// TIA Portal V17 export
// export: Created 2025-03-10T12:15:34.5959597Z, ExportSetting WithDefaults, DisplayName Totally Integrated Automation Portal, DisplayVersion V17 Update 8, DisplayName TIA Portal Openness, DisplayVersion V17 Update 8, DisplayName TIA Portal Version Control Interface, DisplayVersion V17, DisplayName SINAMICS Startdrive Advanced, DisplayVersion V17 SP2, DisplayName SINAMICS Startdrive G110M, G120, G120C, G120D, G120P, G115D, DisplayVersion V17 SP2, DisplayName SINAMICS Startdrive G130, G150, S120, S150, SINAMICS MV, S210, DisplayVersion V17 SP2, DisplayName STEP 7 Professional, DisplayVersion V17 Update 8, DisplayName SINUMERIK ONE STEP 7 Toolbox, DisplayVersion V17 Update 12, DisplayName SINUMERIK 840D sl STEP 7 Toolbox, DisplayVersion V17 Update 12, DisplayName STEP 7 Safety, DisplayVersion V17 Update 6, DisplayName WinCC Advanced, DisplayVersion V17 Update 8
FUNCTION "FC369_NCK_M_CH8_UNIT_03" : Void   // FC369, LAD
TITLE = Channel 1 data
{ S7_Optimized_Access := 'FALSE' }
AUTHOR : ETXETAR
VERSION : 1.0
// stored: AutoNumber false, IsIECCheckEnabled false, SetENOAutomatically false, UDAEnableTagReadback false
BEGIN

REGION Network 1: ACKNOWLEDGE M400-FIXTURE 1 CLAMP SEQUENCE (READ-IN DISABLE) / ACKNOWLEDGE M100-CLAMP SEQUENCE FIXTURE 1
   // NOTE: WHEN THERE IS NOT INDEXING TABLE AVAILABLE IN THE MACHINE DELETE 
   // DB2171.DBX5.0 AND DB2171.DBX2.0
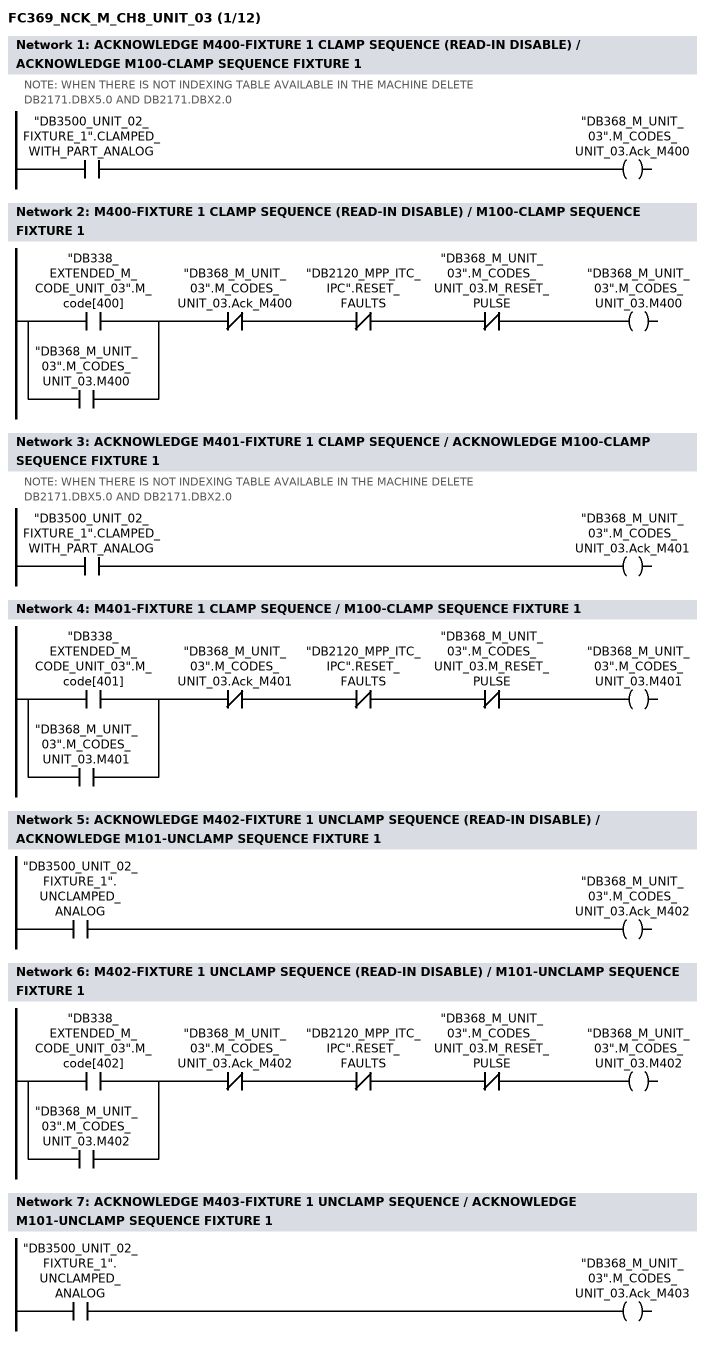
   RUNG wire#powerrail
      Contact( "DB3500_UNIT_02_FIXTURE_1".CLAMPED_WITH_PART_ANALOG )
      Coil( "DB368_M_UNIT_03".M_CODES_UNIT_03.Ack_M400 )
   END_RUNG
   // the same network as SCL:
   "DB368_M_UNIT_03".M_CODES_UNIT_03.Ack_M400 := "DB3500_UNIT_02_FIXTURE_1".CLAMPED_WITH_PART_ANALOG;
END_REGION

REGION Network 2: M400-FIXTURE 1 CLAMP SEQUENCE (READ-IN DISABLE) / M100-CLAMP SEQUENCE FIXTURE 1
   RUNG wire#powerrail
      Contact( "DB338_EXTENDED_M_CODE_UNIT_03".M_code[400] )
      wire#w1
      I_Contact( "DB368_M_UNIT_03".M_CODES_UNIT_03.Ack_M400 )
      I_Contact( "DB2120_MPP_ITC_IPC".RESET_FAULTS )
      I_Contact( "DB368_M_UNIT_03".M_CODES_UNIT_03.M_RESET_PULSE )
      Coil( "DB368_M_UNIT_03".M_CODES_UNIT_03.M400 )
   END_RUNG
   RUNG wire#powerrail
      Contact( "DB368_M_UNIT_03".M_CODES_UNIT_03.M400 )
   END_RUNG wire#w1
   // the same network as SCL:
   "DB368_M_UNIT_03".M_CODES_UNIT_03.M400 := ("DB338_EXTENDED_M_CODE_UNIT_03".M_code[400] OR "DB368_M_UNIT_03".M_CODES_UNIT_03.M400) AND NOT "DB368_M_UNIT_03".M_CODES_UNIT_03.Ack_M400 AND NOT "DB2120_MPP_ITC_IPC".RESET_FAULTS AND NOT "DB368_M_UNIT_03".M_CODES_UNIT_03.M_RESET_PULSE;
END_REGION

REGION Network 3: ACKNOWLEDGE M401-FIXTURE 1 CLAMP SEQUENCE / ACKNOWLEDGE M100-CLAMP SEQUENCE FIXTURE 1
   // NOTE: WHEN THERE IS NOT INDEXING TABLE AVAILABLE IN THE MACHINE DELETE 
   // DB2171.DBX5.0 AND DB2171.DBX2.0
   RUNG wire#powerrail
      Contact( "DB3500_UNIT_02_FIXTURE_1".CLAMPED_WITH_PART_ANALOG )
      Coil( "DB368_M_UNIT_03".M_CODES_UNIT_03.Ack_M401 )
   END_RUNG
   // the same network as SCL:
   "DB368_M_UNIT_03".M_CODES_UNIT_03.Ack_M401 := "DB3500_UNIT_02_FIXTURE_1".CLAMPED_WITH_PART_ANALOG;
END_REGION

REGION Network 4: M401-FIXTURE 1 CLAMP SEQUENCE / M100-CLAMP SEQUENCE FIXTURE 1
   RUNG wire#powerrail
      Contact( "DB338_EXTENDED_M_CODE_UNIT_03".M_code[401] )
      wire#w1
      I_Contact( "DB368_M_UNIT_03".M_CODES_UNIT_03.Ack_M401 )
      I_Contact( "DB2120_MPP_ITC_IPC".RESET_FAULTS )
      I_Contact( "DB368_M_UNIT_03".M_CODES_UNIT_03.M_RESET_PULSE )
      Coil( "DB368_M_UNIT_03".M_CODES_UNIT_03.M401 )
   END_RUNG
   RUNG wire#powerrail
      Contact( "DB368_M_UNIT_03".M_CODES_UNIT_03.M401 )
   END_RUNG wire#w1
   // the same network as SCL:
   "DB368_M_UNIT_03".M_CODES_UNIT_03.M401 := ("DB338_EXTENDED_M_CODE_UNIT_03".M_code[401] OR "DB368_M_UNIT_03".M_CODES_UNIT_03.M401) AND NOT "DB368_M_UNIT_03".M_CODES_UNIT_03.Ack_M401 AND NOT "DB2120_MPP_ITC_IPC".RESET_FAULTS AND NOT "DB368_M_UNIT_03".M_CODES_UNIT_03.M_RESET_PULSE;
END_REGION

REGION Network 5: ACKNOWLEDGE M402-FIXTURE 1 UNCLAMP SEQUENCE (READ-IN DISABLE) / ACKNOWLEDGE M101-UNCLAMP SEQUENCE FIXTURE 1
   RUNG wire#powerrail
      Contact( "DB3500_UNIT_02_FIXTURE_1".UNCLAMPED_ANALOG )
      Coil( "DB368_M_UNIT_03".M_CODES_UNIT_03.Ack_M402 )
   END_RUNG
   // the same network as SCL:
   "DB368_M_UNIT_03".M_CODES_UNIT_03.Ack_M402 := "DB3500_UNIT_02_FIXTURE_1".UNCLAMPED_ANALOG;
END_REGION

REGION Network 6: M402-FIXTURE 1 UNCLAMP SEQUENCE (READ-IN DISABLE) / M101-UNCLAMP SEQUENCE FIXTURE 1
   RUNG wire#powerrail
      Contact( "DB338_EXTENDED_M_CODE_UNIT_03".M_code[402] )
      wire#w1
      I_Contact( "DB368_M_UNIT_03".M_CODES_UNIT_03.Ack_M402 )
      I_Contact( "DB2120_MPP_ITC_IPC".RESET_FAULTS )
      I_Contact( "DB368_M_UNIT_03".M_CODES_UNIT_03.M_RESET_PULSE )
      Coil( "DB368_M_UNIT_03".M_CODES_UNIT_03.M402 )
   END_RUNG
   RUNG wire#powerrail
      Contact( "DB368_M_UNIT_03".M_CODES_UNIT_03.M402 )
   END_RUNG wire#w1
   // the same network as SCL:
   "DB368_M_UNIT_03".M_CODES_UNIT_03.M402 := ("DB338_EXTENDED_M_CODE_UNIT_03".M_code[402] OR "DB368_M_UNIT_03".M_CODES_UNIT_03.M402) AND NOT "DB368_M_UNIT_03".M_CODES_UNIT_03.Ack_M402 AND NOT "DB2120_MPP_ITC_IPC".RESET_FAULTS AND NOT "DB368_M_UNIT_03".M_CODES_UNIT_03.M_RESET_PULSE;
END_REGION

REGION Network 7: ACKNOWLEDGE M403-FIXTURE 1 UNCLAMP SEQUENCE / ACKNOWLEDGE M101-UNCLAMP SEQUENCE FIXTURE 1
   RUNG wire#powerrail
      Contact( "DB3500_UNIT_02_FIXTURE_1".UNCLAMPED_ANALOG )
      Coil( "DB368_M_UNIT_03".M_CODES_UNIT_03.Ack_M403 )
   END_RUNG
   // the same network as SCL:
   "DB368_M_UNIT_03".M_CODES_UNIT_03.Ack_M403 := "DB3500_UNIT_02_FIXTURE_1".UNCLAMPED_ANALOG;
END_REGION

REGION Network 8: M403-FIXTURE 1 UNCLAMP SEQUENCE / M101-UNCLAMP SEQUENCE FIXTURE 1
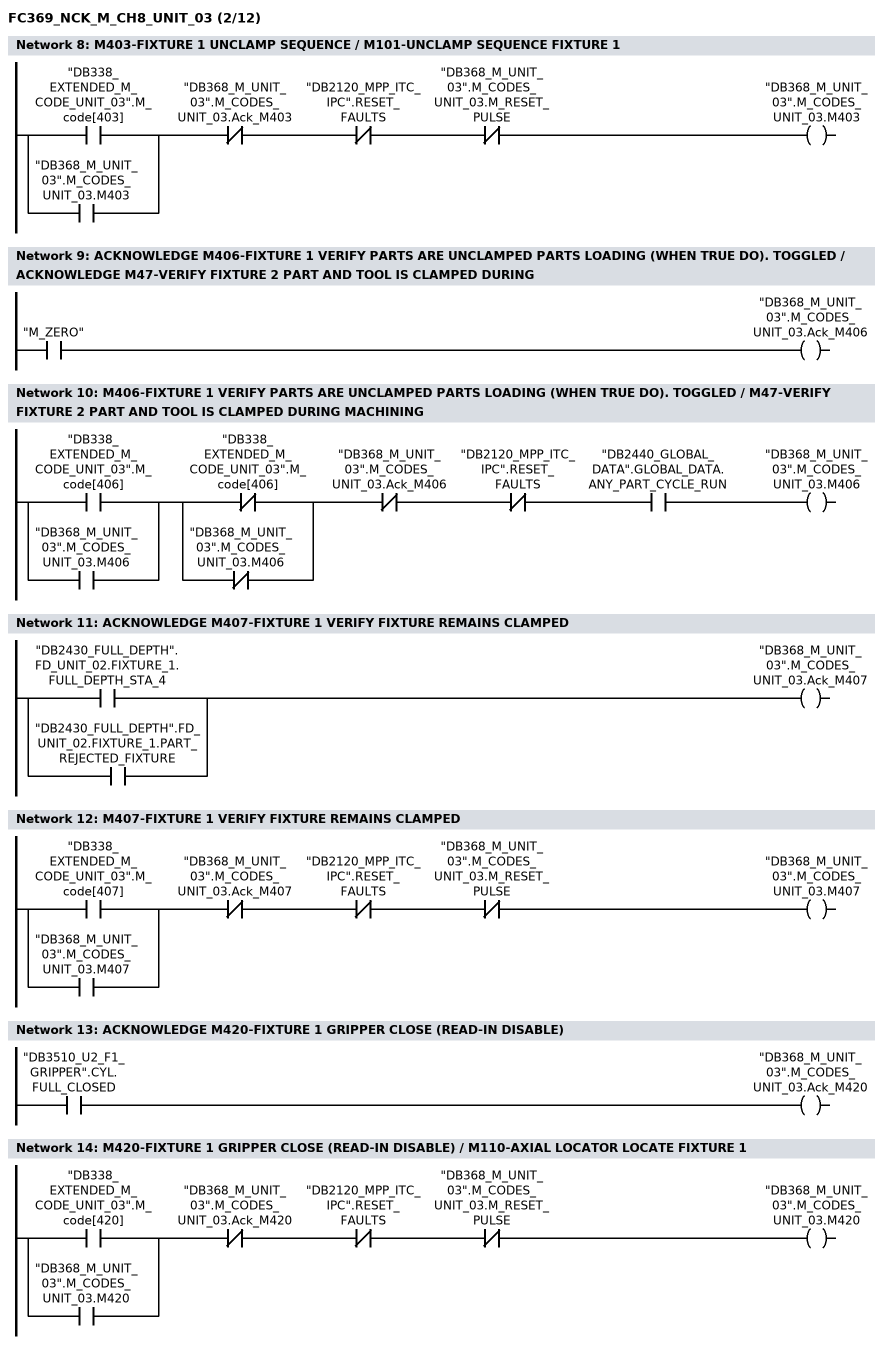
   RUNG wire#powerrail
      Contact( "DB338_EXTENDED_M_CODE_UNIT_03".M_code[403] )
      wire#w1
      I_Contact( "DB368_M_UNIT_03".M_CODES_UNIT_03.Ack_M403 )
      I_Contact( "DB2120_MPP_ITC_IPC".RESET_FAULTS )
      I_Contact( "DB368_M_UNIT_03".M_CODES_UNIT_03.M_RESET_PULSE )
      Coil( "DB368_M_UNIT_03".M_CODES_UNIT_03.M403 )
   END_RUNG
   RUNG wire#powerrail
      Contact( "DB368_M_UNIT_03".M_CODES_UNIT_03.M403 )
   END_RUNG wire#w1
   // the same network as SCL:
   "DB368_M_UNIT_03".M_CODES_UNIT_03.M403 := ("DB338_EXTENDED_M_CODE_UNIT_03".M_code[403] OR "DB368_M_UNIT_03".M_CODES_UNIT_03.M403) AND NOT "DB368_M_UNIT_03".M_CODES_UNIT_03.Ack_M403 AND NOT "DB2120_MPP_ITC_IPC".RESET_FAULTS AND NOT "DB368_M_UNIT_03".M_CODES_UNIT_03.M_RESET_PULSE;
END_REGION

REGION Network 9: ACKNOWLEDGE M406-FIXTURE 1 VERIFY PARTS ARE UNCLAMPED PARTS LOADING (WHEN TRUE DO). TOGGLED / ACKNOWLEDGE M47-VERIFY FIXTURE 2 PART AND TOOL IS CLAMPED DURING
   RUNG wire#powerrail
      Contact( "M_ZERO" )
      Coil( "DB368_M_UNIT_03".M_CODES_UNIT_03.Ack_M406 )
   END_RUNG
   // the same network as SCL:
   "DB368_M_UNIT_03".M_CODES_UNIT_03.Ack_M406 := "M_ZERO";
END_REGION

REGION Network 10: M406-FIXTURE 1 VERIFY PARTS ARE UNCLAMPED PARTS LOADING (WHEN TRUE DO). TOGGLED / M47-VERIFY FIXTURE 2 PART AND TOOL IS CLAMPED DURING MACHINING
   RUNG wire#powerrail
      Contact( "DB338_EXTENDED_M_CODE_UNIT_03".M_code[406] )
      wire#w1
      I_Contact( "DB338_EXTENDED_M_CODE_UNIT_03".M_code[406] )
      wire#w2
      I_Contact( "DB368_M_UNIT_03".M_CODES_UNIT_03.Ack_M406 )
      I_Contact( "DB2120_MPP_ITC_IPC".RESET_FAULTS )
      Contact( "DB2440_GLOBAL_DATA".GLOBAL_DATA.ANY_PART_CYCLE_RUN )
      Coil( "DB368_M_UNIT_03".M_CODES_UNIT_03.M406 )
   END_RUNG
   RUNG wire#powerrail
      Contact( "DB368_M_UNIT_03".M_CODES_UNIT_03.M406 )
   END_RUNG wire#w1
   RUNG wire#w1
      I_Contact( "DB368_M_UNIT_03".M_CODES_UNIT_03.M406 )
   END_RUNG wire#w2
   // the same network as SCL:
   "DB368_M_UNIT_03".M_CODES_UNIT_03.M406 := ("DB338_EXTENDED_M_CODE_UNIT_03".M_code[406] OR "DB368_M_UNIT_03".M_CODES_UNIT_03.M406) AND (NOT "DB338_EXTENDED_M_CODE_UNIT_03".M_code[406] OR NOT "DB368_M_UNIT_03".M_CODES_UNIT_03.M406) AND NOT "DB368_M_UNIT_03".M_CODES_UNIT_03.Ack_M406 AND NOT "DB2120_MPP_ITC_IPC".RESET_FAULTS AND "DB2440_GLOBAL_DATA".GLOBAL_DATA.ANY_PART_CYCLE_RUN;
END_REGION

REGION Network 11: ACKNOWLEDGE M407-FIXTURE 1 VERIFY FIXTURE REMAINS CLAMPED
   RUNG wire#powerrail
      Contact( "DB2430_FULL_DEPTH".FD_UNIT_02.FIXTURE_1.FULL_DEPTH_STA_4 )
      wire#w1
      Coil( "DB368_M_UNIT_03".M_CODES_UNIT_03.Ack_M407 )
   END_RUNG
   RUNG wire#powerrail
      Contact( "DB2430_FULL_DEPTH".FD_UNIT_02.FIXTURE_1.PART_REJECTED_FIXTURE )
   END_RUNG wire#w1
   // the same network as SCL:
   "DB368_M_UNIT_03".M_CODES_UNIT_03.Ack_M407 := "DB2430_FULL_DEPTH".FD_UNIT_02.FIXTURE_1.FULL_DEPTH_STA_4 OR "DB2430_FULL_DEPTH".FD_UNIT_02.FIXTURE_1.PART_REJECTED_FIXTURE;
END_REGION

REGION Network 12: M407-FIXTURE 1 VERIFY FIXTURE REMAINS CLAMPED
   RUNG wire#powerrail
      Contact( "DB338_EXTENDED_M_CODE_UNIT_03".M_code[407] )
      wire#w1
      I_Contact( "DB368_M_UNIT_03".M_CODES_UNIT_03.Ack_M407 )
      I_Contact( "DB2120_MPP_ITC_IPC".RESET_FAULTS )
      I_Contact( "DB368_M_UNIT_03".M_CODES_UNIT_03.M_RESET_PULSE )
      Coil( "DB368_M_UNIT_03".M_CODES_UNIT_03.M407 )
   END_RUNG
   RUNG wire#powerrail
      Contact( "DB368_M_UNIT_03".M_CODES_UNIT_03.M407 )
   END_RUNG wire#w1
   // the same network as SCL:
   "DB368_M_UNIT_03".M_CODES_UNIT_03.M407 := ("DB338_EXTENDED_M_CODE_UNIT_03".M_code[407] OR "DB368_M_UNIT_03".M_CODES_UNIT_03.M407) AND NOT "DB368_M_UNIT_03".M_CODES_UNIT_03.Ack_M407 AND NOT "DB2120_MPP_ITC_IPC".RESET_FAULTS AND NOT "DB368_M_UNIT_03".M_CODES_UNIT_03.M_RESET_PULSE;
END_REGION

REGION Network 13: ACKNOWLEDGE M420-FIXTURE 1 GRIPPER CLOSE (READ-IN DISABLE)
   RUNG wire#powerrail
      Contact( "DB3510_U2_F1_GRIPPER".CYL.FULL_CLOSED )
      Coil( "DB368_M_UNIT_03".M_CODES_UNIT_03.Ack_M420 )
   END_RUNG
   // the same network as SCL:
   "DB368_M_UNIT_03".M_CODES_UNIT_03.Ack_M420 := "DB3510_U2_F1_GRIPPER".CYL.FULL_CLOSED;
END_REGION

REGION Network 14: M420-FIXTURE 1 GRIPPER CLOSE (READ-IN DISABLE) / M110-AXIAL LOCATOR LOCATE FIXTURE 1
   RUNG wire#powerrail
      Contact( "DB338_EXTENDED_M_CODE_UNIT_03".M_code[420] )
      wire#w1
      I_Contact( "DB368_M_UNIT_03".M_CODES_UNIT_03.Ack_M420 )
      I_Contact( "DB2120_MPP_ITC_IPC".RESET_FAULTS )
      I_Contact( "DB368_M_UNIT_03".M_CODES_UNIT_03.M_RESET_PULSE )
      Coil( "DB368_M_UNIT_03".M_CODES_UNIT_03.M420 )
   END_RUNG
   RUNG wire#powerrail
      Contact( "DB368_M_UNIT_03".M_CODES_UNIT_03.M420 )
   END_RUNG wire#w1
   // the same network as SCL:
   "DB368_M_UNIT_03".M_CODES_UNIT_03.M420 := ("DB338_EXTENDED_M_CODE_UNIT_03".M_code[420] OR "DB368_M_UNIT_03".M_CODES_UNIT_03.M420) AND NOT "DB368_M_UNIT_03".M_CODES_UNIT_03.Ack_M420 AND NOT "DB2120_MPP_ITC_IPC".RESET_FAULTS AND NOT "DB368_M_UNIT_03".M_CODES_UNIT_03.M_RESET_PULSE;
END_REGION

REGION Network 15: ACKNOWLEDGE M421-FIXTURE 1 GRIPPER CLOSE
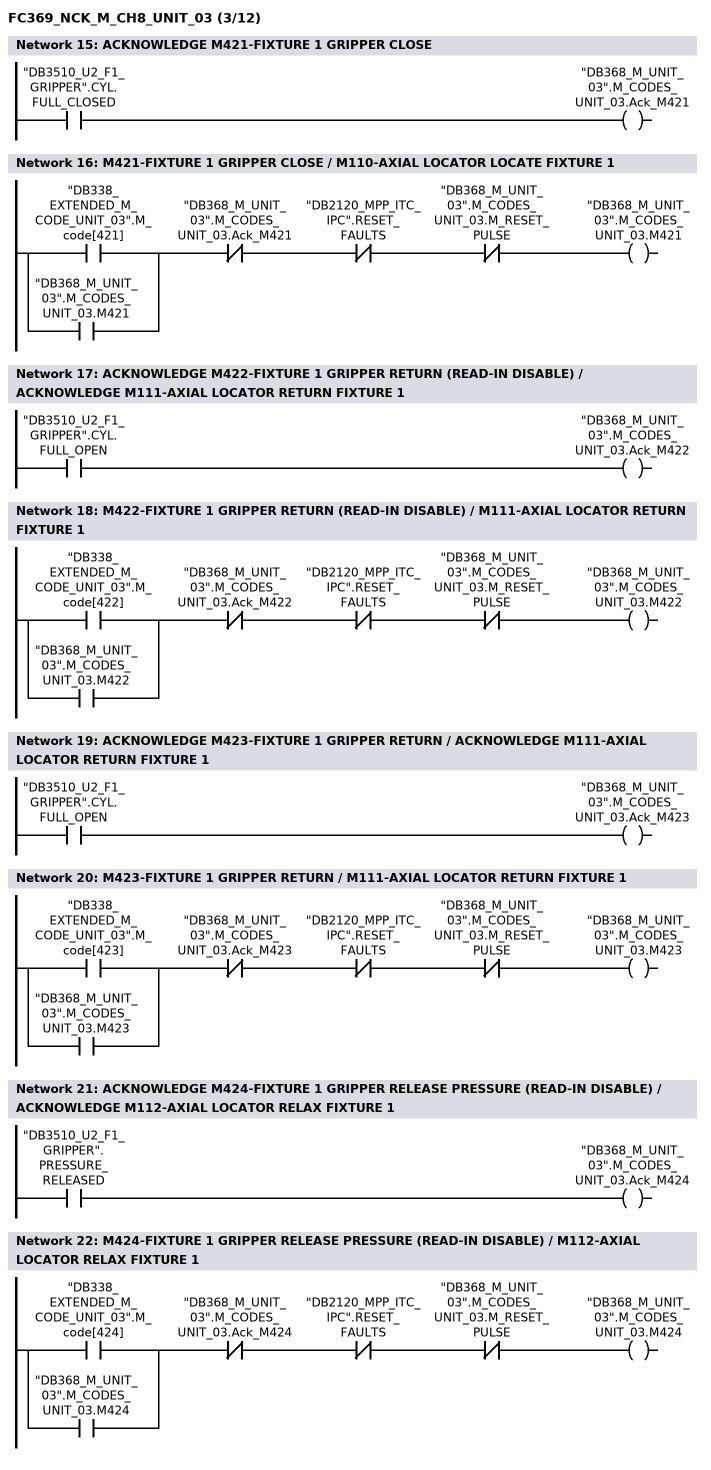
   RUNG wire#powerrail
      Contact( "DB3510_U2_F1_GRIPPER".CYL.FULL_CLOSED )
      Coil( "DB368_M_UNIT_03".M_CODES_UNIT_03.Ack_M421 )
   END_RUNG
   // the same network as SCL:
   "DB368_M_UNIT_03".M_CODES_UNIT_03.Ack_M421 := "DB3510_U2_F1_GRIPPER".CYL.FULL_CLOSED;
END_REGION

REGION Network 16: M421-FIXTURE 1 GRIPPER CLOSE / M110-AXIAL LOCATOR LOCATE FIXTURE 1
   RUNG wire#powerrail
      Contact( "DB338_EXTENDED_M_CODE_UNIT_03".M_code[421] )
      wire#w1
      I_Contact( "DB368_M_UNIT_03".M_CODES_UNIT_03.Ack_M421 )
      I_Contact( "DB2120_MPP_ITC_IPC".RESET_FAULTS )
      I_Contact( "DB368_M_UNIT_03".M_CODES_UNIT_03.M_RESET_PULSE )
      Coil( "DB368_M_UNIT_03".M_CODES_UNIT_03.M421 )
   END_RUNG
   RUNG wire#powerrail
      Contact( "DB368_M_UNIT_03".M_CODES_UNIT_03.M421 )
   END_RUNG wire#w1
   // the same network as SCL:
   "DB368_M_UNIT_03".M_CODES_UNIT_03.M421 := ("DB338_EXTENDED_M_CODE_UNIT_03".M_code[421] OR "DB368_M_UNIT_03".M_CODES_UNIT_03.M421) AND NOT "DB368_M_UNIT_03".M_CODES_UNIT_03.Ack_M421 AND NOT "DB2120_MPP_ITC_IPC".RESET_FAULTS AND NOT "DB368_M_UNIT_03".M_CODES_UNIT_03.M_RESET_PULSE;
END_REGION

REGION Network 17: ACKNOWLEDGE M422-FIXTURE 1 GRIPPER RETURN (READ-IN DISABLE) / ACKNOWLEDGE M111-AXIAL LOCATOR RETURN FIXTURE 1
   RUNG wire#powerrail
      Contact( "DB3510_U2_F1_GRIPPER".CYL.FULL_OPEN )
      Coil( "DB368_M_UNIT_03".M_CODES_UNIT_03.Ack_M422 )
   END_RUNG
   // the same network as SCL:
   "DB368_M_UNIT_03".M_CODES_UNIT_03.Ack_M422 := "DB3510_U2_F1_GRIPPER".CYL.FULL_OPEN;
END_REGION

REGION Network 18: M422-FIXTURE 1 GRIPPER RETURN (READ-IN DISABLE) / M111-AXIAL LOCATOR RETURN FIXTURE 1
   RUNG wire#powerrail
      Contact( "DB338_EXTENDED_M_CODE_UNIT_03".M_code[422] )
      wire#w1
      I_Contact( "DB368_M_UNIT_03".M_CODES_UNIT_03.Ack_M422 )
      I_Contact( "DB2120_MPP_ITC_IPC".RESET_FAULTS )
      I_Contact( "DB368_M_UNIT_03".M_CODES_UNIT_03.M_RESET_PULSE )
      Coil( "DB368_M_UNIT_03".M_CODES_UNIT_03.M422 )
   END_RUNG
   RUNG wire#powerrail
      Contact( "DB368_M_UNIT_03".M_CODES_UNIT_03.M422 )
   END_RUNG wire#w1
   // the same network as SCL:
   "DB368_M_UNIT_03".M_CODES_UNIT_03.M422 := ("DB338_EXTENDED_M_CODE_UNIT_03".M_code[422] OR "DB368_M_UNIT_03".M_CODES_UNIT_03.M422) AND NOT "DB368_M_UNIT_03".M_CODES_UNIT_03.Ack_M422 AND NOT "DB2120_MPP_ITC_IPC".RESET_FAULTS AND NOT "DB368_M_UNIT_03".M_CODES_UNIT_03.M_RESET_PULSE;
END_REGION

REGION Network 19: ACKNOWLEDGE M423-FIXTURE 1 GRIPPER RETURN / ACKNOWLEDGE M111-AXIAL LOCATOR RETURN FIXTURE 1
   RUNG wire#powerrail
      Contact( "DB3510_U2_F1_GRIPPER".CYL.FULL_OPEN )
      Coil( "DB368_M_UNIT_03".M_CODES_UNIT_03.Ack_M423 )
   END_RUNG
   // the same network as SCL:
   "DB368_M_UNIT_03".M_CODES_UNIT_03.Ack_M423 := "DB3510_U2_F1_GRIPPER".CYL.FULL_OPEN;
END_REGION

REGION Network 20: M423-FIXTURE 1 GRIPPER RETURN / M111-AXIAL LOCATOR RETURN FIXTURE 1
   RUNG wire#powerrail
      Contact( "DB338_EXTENDED_M_CODE_UNIT_03".M_code[423] )
      wire#w1
      I_Contact( "DB368_M_UNIT_03".M_CODES_UNIT_03.Ack_M423 )
      I_Contact( "DB2120_MPP_ITC_IPC".RESET_FAULTS )
      I_Contact( "DB368_M_UNIT_03".M_CODES_UNIT_03.M_RESET_PULSE )
      Coil( "DB368_M_UNIT_03".M_CODES_UNIT_03.M423 )
   END_RUNG
   RUNG wire#powerrail
      Contact( "DB368_M_UNIT_03".M_CODES_UNIT_03.M423 )
   END_RUNG wire#w1
   // the same network as SCL:
   "DB368_M_UNIT_03".M_CODES_UNIT_03.M423 := ("DB338_EXTENDED_M_CODE_UNIT_03".M_code[423] OR "DB368_M_UNIT_03".M_CODES_UNIT_03.M423) AND NOT "DB368_M_UNIT_03".M_CODES_UNIT_03.Ack_M423 AND NOT "DB2120_MPP_ITC_IPC".RESET_FAULTS AND NOT "DB368_M_UNIT_03".M_CODES_UNIT_03.M_RESET_PULSE;
END_REGION

REGION Network 21: ACKNOWLEDGE M424-FIXTURE 1 GRIPPER RELEASE PRESSURE (READ-IN DISABLE) / ACKNOWLEDGE M112-AXIAL LOCATOR RELAX FIXTURE 1
   RUNG wire#powerrail
      Contact( "DB3510_U2_F1_GRIPPER".PRESSURE_RELEASED )
      Coil( "DB368_M_UNIT_03".M_CODES_UNIT_03.Ack_M424 )
   END_RUNG
   // the same network as SCL:
   "DB368_M_UNIT_03".M_CODES_UNIT_03.Ack_M424 := "DB3510_U2_F1_GRIPPER".PRESSURE_RELEASED;
END_REGION

REGION Network 22: M424-FIXTURE 1 GRIPPER RELEASE PRESSURE (READ-IN DISABLE) / M112-AXIAL LOCATOR RELAX FIXTURE 1
   RUNG wire#powerrail
      Contact( "DB338_EXTENDED_M_CODE_UNIT_03".M_code[424] )
      wire#w1
      I_Contact( "DB368_M_UNIT_03".M_CODES_UNIT_03.Ack_M424 )
      I_Contact( "DB2120_MPP_ITC_IPC".RESET_FAULTS )
      I_Contact( "DB368_M_UNIT_03".M_CODES_UNIT_03.M_RESET_PULSE )
      Coil( "DB368_M_UNIT_03".M_CODES_UNIT_03.M424 )
   END_RUNG
   RUNG wire#powerrail
      Contact( "DB368_M_UNIT_03".M_CODES_UNIT_03.M424 )
   END_RUNG wire#w1
   // the same network as SCL:
   "DB368_M_UNIT_03".M_CODES_UNIT_03.M424 := ("DB338_EXTENDED_M_CODE_UNIT_03".M_code[424] OR "DB368_M_UNIT_03".M_CODES_UNIT_03.M424) AND NOT "DB368_M_UNIT_03".M_CODES_UNIT_03.Ack_M424 AND NOT "DB2120_MPP_ITC_IPC".RESET_FAULTS AND NOT "DB368_M_UNIT_03".M_CODES_UNIT_03.M_RESET_PULSE;
END_REGION

REGION Network 23: ACKNOWLEDGE M425-FIXTURE 1 GRIPPER LOW PRESSURE (READ-IN DISABLE) / ACKNOWLEDGE M23-SWITCH ON SPINDLE FRAME BLOWING
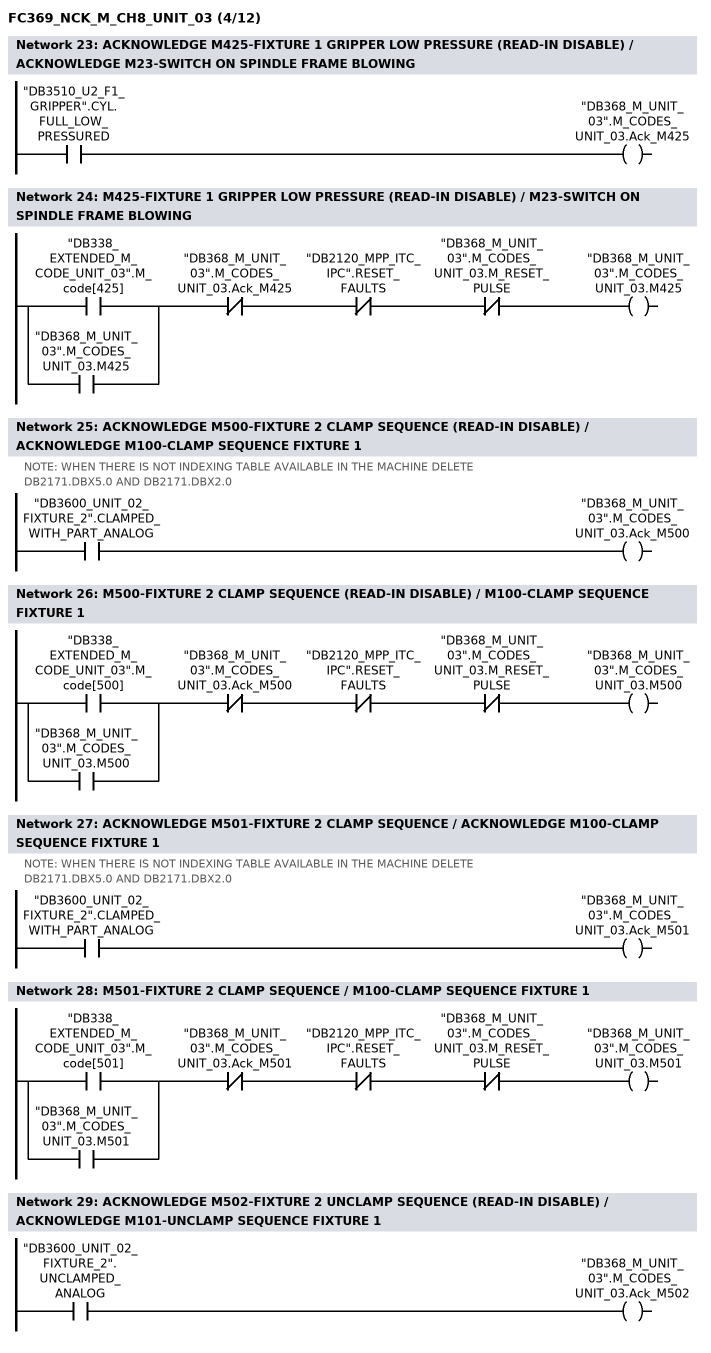
   RUNG wire#powerrail
      Contact( "DB3510_U2_F1_GRIPPER".CYL.FULL_LOW_PRESSURED )
      Coil( "DB368_M_UNIT_03".M_CODES_UNIT_03.Ack_M425 )
   END_RUNG
   // the same network as SCL:
   "DB368_M_UNIT_03".M_CODES_UNIT_03.Ack_M425 := "DB3510_U2_F1_GRIPPER".CYL.FULL_LOW_PRESSURED;
END_REGION

REGION Network 24: M425-FIXTURE 1 GRIPPER LOW PRESSURE (READ-IN DISABLE) / M23-SWITCH ON SPINDLE FRAME BLOWING
   RUNG wire#powerrail
      Contact( "DB338_EXTENDED_M_CODE_UNIT_03".M_code[425] )
      wire#w1
      I_Contact( "DB368_M_UNIT_03".M_CODES_UNIT_03.Ack_M425 )
      I_Contact( "DB2120_MPP_ITC_IPC".RESET_FAULTS )
      I_Contact( "DB368_M_UNIT_03".M_CODES_UNIT_03.M_RESET_PULSE )
      Coil( "DB368_M_UNIT_03".M_CODES_UNIT_03.M425 )
   END_RUNG
   RUNG wire#powerrail
      Contact( "DB368_M_UNIT_03".M_CODES_UNIT_03.M425 )
   END_RUNG wire#w1
   // the same network as SCL:
   "DB368_M_UNIT_03".M_CODES_UNIT_03.M425 := ("DB338_EXTENDED_M_CODE_UNIT_03".M_code[425] OR "DB368_M_UNIT_03".M_CODES_UNIT_03.M425) AND NOT "DB368_M_UNIT_03".M_CODES_UNIT_03.Ack_M425 AND NOT "DB2120_MPP_ITC_IPC".RESET_FAULTS AND NOT "DB368_M_UNIT_03".M_CODES_UNIT_03.M_RESET_PULSE;
END_REGION

REGION Network 25: ACKNOWLEDGE M500-FIXTURE 2 CLAMP SEQUENCE (READ-IN DISABLE) / ACKNOWLEDGE M100-CLAMP SEQUENCE FIXTURE 1
   // NOTE: WHEN THERE IS NOT INDEXING TABLE AVAILABLE IN THE MACHINE DELETE 
   // DB2171.DBX5.0 AND DB2171.DBX2.0
   RUNG wire#powerrail
      Contact( "DB3600_UNIT_02_FIXTURE_2".CLAMPED_WITH_PART_ANALOG )
      Coil( "DB368_M_UNIT_03".M_CODES_UNIT_03.Ack_M500 )
   END_RUNG
   // the same network as SCL:
   "DB368_M_UNIT_03".M_CODES_UNIT_03.Ack_M500 := "DB3600_UNIT_02_FIXTURE_2".CLAMPED_WITH_PART_ANALOG;
END_REGION

REGION Network 26: M500-FIXTURE 2 CLAMP SEQUENCE (READ-IN DISABLE) / M100-CLAMP SEQUENCE FIXTURE 1
   RUNG wire#powerrail
      Contact( "DB338_EXTENDED_M_CODE_UNIT_03".M_code[500] )
      wire#w1
      I_Contact( "DB368_M_UNIT_03".M_CODES_UNIT_03.Ack_M500 )
      I_Contact( "DB2120_MPP_ITC_IPC".RESET_FAULTS )
      I_Contact( "DB368_M_UNIT_03".M_CODES_UNIT_03.M_RESET_PULSE )
      Coil( "DB368_M_UNIT_03".M_CODES_UNIT_03.M500 )
   END_RUNG
   RUNG wire#powerrail
      Contact( "DB368_M_UNIT_03".M_CODES_UNIT_03.M500 )
   END_RUNG wire#w1
   // the same network as SCL:
   "DB368_M_UNIT_03".M_CODES_UNIT_03.M500 := ("DB338_EXTENDED_M_CODE_UNIT_03".M_code[500] OR "DB368_M_UNIT_03".M_CODES_UNIT_03.M500) AND NOT "DB368_M_UNIT_03".M_CODES_UNIT_03.Ack_M500 AND NOT "DB2120_MPP_ITC_IPC".RESET_FAULTS AND NOT "DB368_M_UNIT_03".M_CODES_UNIT_03.M_RESET_PULSE;
END_REGION

REGION Network 27: ACKNOWLEDGE M501-FIXTURE 2 CLAMP SEQUENCE / ACKNOWLEDGE M100-CLAMP SEQUENCE FIXTURE 1
   // NOTE: WHEN THERE IS NOT INDEXING TABLE AVAILABLE IN THE MACHINE DELETE 
   // DB2171.DBX5.0 AND DB2171.DBX2.0
   RUNG wire#powerrail
      Contact( "DB3600_UNIT_02_FIXTURE_2".CLAMPED_WITH_PART_ANALOG )
      Coil( "DB368_M_UNIT_03".M_CODES_UNIT_03.Ack_M501 )
   END_RUNG
   // the same network as SCL:
   "DB368_M_UNIT_03".M_CODES_UNIT_03.Ack_M501 := "DB3600_UNIT_02_FIXTURE_2".CLAMPED_WITH_PART_ANALOG;
END_REGION

REGION Network 28: M501-FIXTURE 2 CLAMP SEQUENCE / M100-CLAMP SEQUENCE FIXTURE 1
   RUNG wire#powerrail
      Contact( "DB338_EXTENDED_M_CODE_UNIT_03".M_code[501] )
      wire#w1
      I_Contact( "DB368_M_UNIT_03".M_CODES_UNIT_03.Ack_M501 )
      I_Contact( "DB2120_MPP_ITC_IPC".RESET_FAULTS )
      I_Contact( "DB368_M_UNIT_03".M_CODES_UNIT_03.M_RESET_PULSE )
      Coil( "DB368_M_UNIT_03".M_CODES_UNIT_03.M501 )
   END_RUNG
   RUNG wire#powerrail
      Contact( "DB368_M_UNIT_03".M_CODES_UNIT_03.M501 )
   END_RUNG wire#w1
   // the same network as SCL:
   "DB368_M_UNIT_03".M_CODES_UNIT_03.M501 := ("DB338_EXTENDED_M_CODE_UNIT_03".M_code[501] OR "DB368_M_UNIT_03".M_CODES_UNIT_03.M501) AND NOT "DB368_M_UNIT_03".M_CODES_UNIT_03.Ack_M501 AND NOT "DB2120_MPP_ITC_IPC".RESET_FAULTS AND NOT "DB368_M_UNIT_03".M_CODES_UNIT_03.M_RESET_PULSE;
END_REGION

REGION Network 29: ACKNOWLEDGE M502-FIXTURE 2 UNCLAMP SEQUENCE (READ-IN DISABLE) / ACKNOWLEDGE M101-UNCLAMP SEQUENCE FIXTURE 1
   RUNG wire#powerrail
      Contact( "DB3600_UNIT_02_FIXTURE_2".UNCLAMPED_ANALOG )
      Coil( "DB368_M_UNIT_03".M_CODES_UNIT_03.Ack_M502 )
   END_RUNG
   // the same network as SCL:
   "DB368_M_UNIT_03".M_CODES_UNIT_03.Ack_M502 := "DB3600_UNIT_02_FIXTURE_2".UNCLAMPED_ANALOG;
END_REGION

REGION Network 30: M502-FIXTURE 2 UNCLAMP SEQUENCE (READ-IN DISABLE) / M101-UNCLAMP SEQUENCE FIXTURE 1
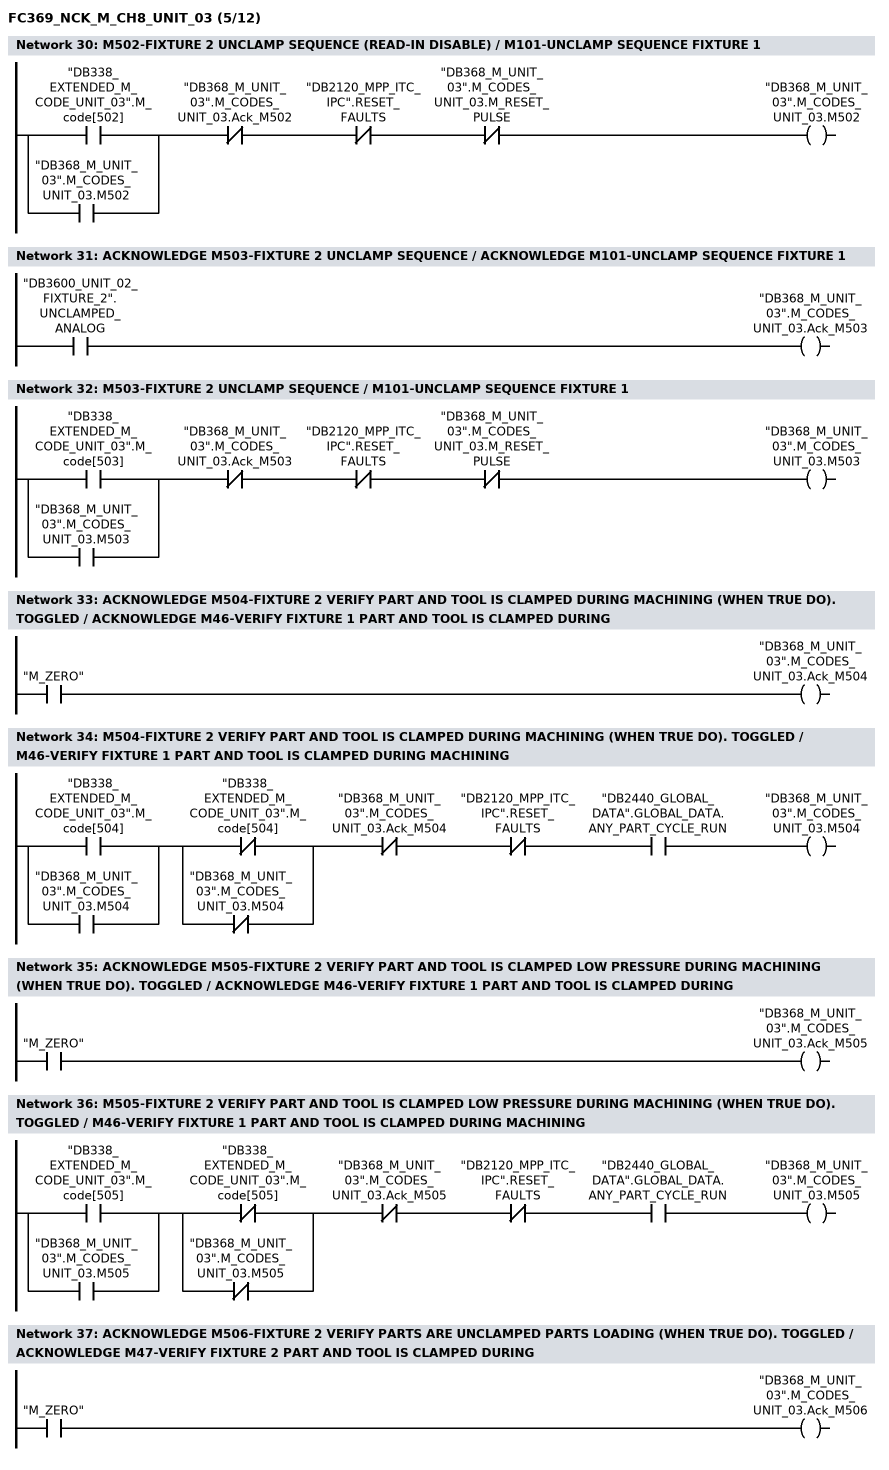
   RUNG wire#powerrail
      Contact( "DB338_EXTENDED_M_CODE_UNIT_03".M_code[502] )
      wire#w1
      I_Contact( "DB368_M_UNIT_03".M_CODES_UNIT_03.Ack_M502 )
      I_Contact( "DB2120_MPP_ITC_IPC".RESET_FAULTS )
      I_Contact( "DB368_M_UNIT_03".M_CODES_UNIT_03.M_RESET_PULSE )
      Coil( "DB368_M_UNIT_03".M_CODES_UNIT_03.M502 )
   END_RUNG
   RUNG wire#powerrail
      Contact( "DB368_M_UNIT_03".M_CODES_UNIT_03.M502 )
   END_RUNG wire#w1
   // the same network as SCL:
   "DB368_M_UNIT_03".M_CODES_UNIT_03.M502 := ("DB338_EXTENDED_M_CODE_UNIT_03".M_code[502] OR "DB368_M_UNIT_03".M_CODES_UNIT_03.M502) AND NOT "DB368_M_UNIT_03".M_CODES_UNIT_03.Ack_M502 AND NOT "DB2120_MPP_ITC_IPC".RESET_FAULTS AND NOT "DB368_M_UNIT_03".M_CODES_UNIT_03.M_RESET_PULSE;
END_REGION

REGION Network 31: ACKNOWLEDGE M503-FIXTURE 2 UNCLAMP SEQUENCE / ACKNOWLEDGE M101-UNCLAMP SEQUENCE FIXTURE 1
   RUNG wire#powerrail
      Contact( "DB3600_UNIT_02_FIXTURE_2".UNCLAMPED_ANALOG )
      Coil( "DB368_M_UNIT_03".M_CODES_UNIT_03.Ack_M503 )
   END_RUNG
   // the same network as SCL:
   "DB368_M_UNIT_03".M_CODES_UNIT_03.Ack_M503 := "DB3600_UNIT_02_FIXTURE_2".UNCLAMPED_ANALOG;
END_REGION

REGION Network 32: M503-FIXTURE 2 UNCLAMP SEQUENCE / M101-UNCLAMP SEQUENCE FIXTURE 1
   RUNG wire#powerrail
      Contact( "DB338_EXTENDED_M_CODE_UNIT_03".M_code[503] )
      wire#w1
      I_Contact( "DB368_M_UNIT_03".M_CODES_UNIT_03.Ack_M503 )
      I_Contact( "DB2120_MPP_ITC_IPC".RESET_FAULTS )
      I_Contact( "DB368_M_UNIT_03".M_CODES_UNIT_03.M_RESET_PULSE )
      Coil( "DB368_M_UNIT_03".M_CODES_UNIT_03.M503 )
   END_RUNG
   RUNG wire#powerrail
      Contact( "DB368_M_UNIT_03".M_CODES_UNIT_03.M503 )
   END_RUNG wire#w1
   // the same network as SCL:
   "DB368_M_UNIT_03".M_CODES_UNIT_03.M503 := ("DB338_EXTENDED_M_CODE_UNIT_03".M_code[503] OR "DB368_M_UNIT_03".M_CODES_UNIT_03.M503) AND NOT "DB368_M_UNIT_03".M_CODES_UNIT_03.Ack_M503 AND NOT "DB2120_MPP_ITC_IPC".RESET_FAULTS AND NOT "DB368_M_UNIT_03".M_CODES_UNIT_03.M_RESET_PULSE;
END_REGION

REGION Network 33: ACKNOWLEDGE M504-FIXTURE 2 VERIFY PART AND TOOL IS CLAMPED DURING MACHINING (WHEN TRUE DO). TOGGLED / ACKNOWLEDGE M46-VERIFY FIXTURE 1 PART AND TOOL IS CLAMPED DURING
   RUNG wire#powerrail
      Contact( "M_ZERO" )
      Coil( "DB368_M_UNIT_03".M_CODES_UNIT_03.Ack_M504 )
   END_RUNG
   // the same network as SCL:
   "DB368_M_UNIT_03".M_CODES_UNIT_03.Ack_M504 := "M_ZERO";
END_REGION

REGION Network 34: M504-FIXTURE 2 VERIFY PART AND TOOL IS CLAMPED DURING MACHINING (WHEN TRUE DO). TOGGLED / M46-VERIFY FIXTURE 1 PART AND TOOL IS CLAMPED DURING MACHINING
   RUNG wire#powerrail
      Contact( "DB338_EXTENDED_M_CODE_UNIT_03".M_code[504] )
      wire#w1
      I_Contact( "DB338_EXTENDED_M_CODE_UNIT_03".M_code[504] )
      wire#w2
      I_Contact( "DB368_M_UNIT_03".M_CODES_UNIT_03.Ack_M504 )
      I_Contact( "DB2120_MPP_ITC_IPC".RESET_FAULTS )
      Contact( "DB2440_GLOBAL_DATA".GLOBAL_DATA.ANY_PART_CYCLE_RUN )
      Coil( "DB368_M_UNIT_03".M_CODES_UNIT_03.M504 )
   END_RUNG
   RUNG wire#powerrail
      Contact( "DB368_M_UNIT_03".M_CODES_UNIT_03.M504 )
   END_RUNG wire#w1
   RUNG wire#w1
      I_Contact( "DB368_M_UNIT_03".M_CODES_UNIT_03.M504 )
   END_RUNG wire#w2
   // the same network as SCL:
   "DB368_M_UNIT_03".M_CODES_UNIT_03.M504 := ("DB338_EXTENDED_M_CODE_UNIT_03".M_code[504] OR "DB368_M_UNIT_03".M_CODES_UNIT_03.M504) AND (NOT "DB338_EXTENDED_M_CODE_UNIT_03".M_code[504] OR NOT "DB368_M_UNIT_03".M_CODES_UNIT_03.M504) AND NOT "DB368_M_UNIT_03".M_CODES_UNIT_03.Ack_M504 AND NOT "DB2120_MPP_ITC_IPC".RESET_FAULTS AND "DB2440_GLOBAL_DATA".GLOBAL_DATA.ANY_PART_CYCLE_RUN;
END_REGION

REGION Network 35: ACKNOWLEDGE M505-FIXTURE 2 VERIFY PART AND TOOL IS CLAMPED LOW PRESSURE DURING MACHINING (WHEN TRUE DO). TOGGLED / ACKNOWLEDGE M46-VERIFY FIXTURE 1 PART AND TOOL IS CLAMPED DURING
   RUNG wire#powerrail
      Contact( "M_ZERO" )
      Coil( "DB368_M_UNIT_03".M_CODES_UNIT_03.Ack_M505 )
   END_RUNG
   // the same network as SCL:
   "DB368_M_UNIT_03".M_CODES_UNIT_03.Ack_M505 := "M_ZERO";
END_REGION

REGION Network 36: M505-FIXTURE 2 VERIFY PART AND TOOL IS CLAMPED LOW PRESSURE DURING MACHINING (WHEN TRUE DO). TOGGLED / M46-VERIFY FIXTURE 1 PART AND TOOL IS CLAMPED DURING MACHINING
   RUNG wire#powerrail
      Contact( "DB338_EXTENDED_M_CODE_UNIT_03".M_code[505] )
      wire#w1
      I_Contact( "DB338_EXTENDED_M_CODE_UNIT_03".M_code[505] )
      wire#w2
      I_Contact( "DB368_M_UNIT_03".M_CODES_UNIT_03.Ack_M505 )
      I_Contact( "DB2120_MPP_ITC_IPC".RESET_FAULTS )
      Contact( "DB2440_GLOBAL_DATA".GLOBAL_DATA.ANY_PART_CYCLE_RUN )
      Coil( "DB368_M_UNIT_03".M_CODES_UNIT_03.M505 )
   END_RUNG
   RUNG wire#powerrail
      Contact( "DB368_M_UNIT_03".M_CODES_UNIT_03.M505 )
   END_RUNG wire#w1
   RUNG wire#w1
      I_Contact( "DB368_M_UNIT_03".M_CODES_UNIT_03.M505 )
   END_RUNG wire#w2
   // the same network as SCL:
   "DB368_M_UNIT_03".M_CODES_UNIT_03.M505 := ("DB338_EXTENDED_M_CODE_UNIT_03".M_code[505] OR "DB368_M_UNIT_03".M_CODES_UNIT_03.M505) AND (NOT "DB338_EXTENDED_M_CODE_UNIT_03".M_code[505] OR NOT "DB368_M_UNIT_03".M_CODES_UNIT_03.M505) AND NOT "DB368_M_UNIT_03".M_CODES_UNIT_03.Ack_M505 AND NOT "DB2120_MPP_ITC_IPC".RESET_FAULTS AND "DB2440_GLOBAL_DATA".GLOBAL_DATA.ANY_PART_CYCLE_RUN;
END_REGION

REGION Network 37: ACKNOWLEDGE M506-FIXTURE 2 VERIFY PARTS ARE UNCLAMPED PARTS LOADING (WHEN TRUE DO). TOGGLED / ACKNOWLEDGE M47-VERIFY FIXTURE 2 PART AND TOOL IS CLAMPED DURING
   RUNG wire#powerrail
      Contact( "M_ZERO" )
      Coil( "DB368_M_UNIT_03".M_CODES_UNIT_03.Ack_M506 )
   END_RUNG
   // the same network as SCL:
   "DB368_M_UNIT_03".M_CODES_UNIT_03.Ack_M506 := "M_ZERO";
END_REGION

REGION Network 38: M506-FIXTURE 2 VERIFY PARTS ARE UNCLAMPED PARTS LOADING (WHEN TRUE DO). TOGGLED / M47-VERIFY FIXTURE 2 PART AND TOOL IS CLAMPED DURING MACHINING
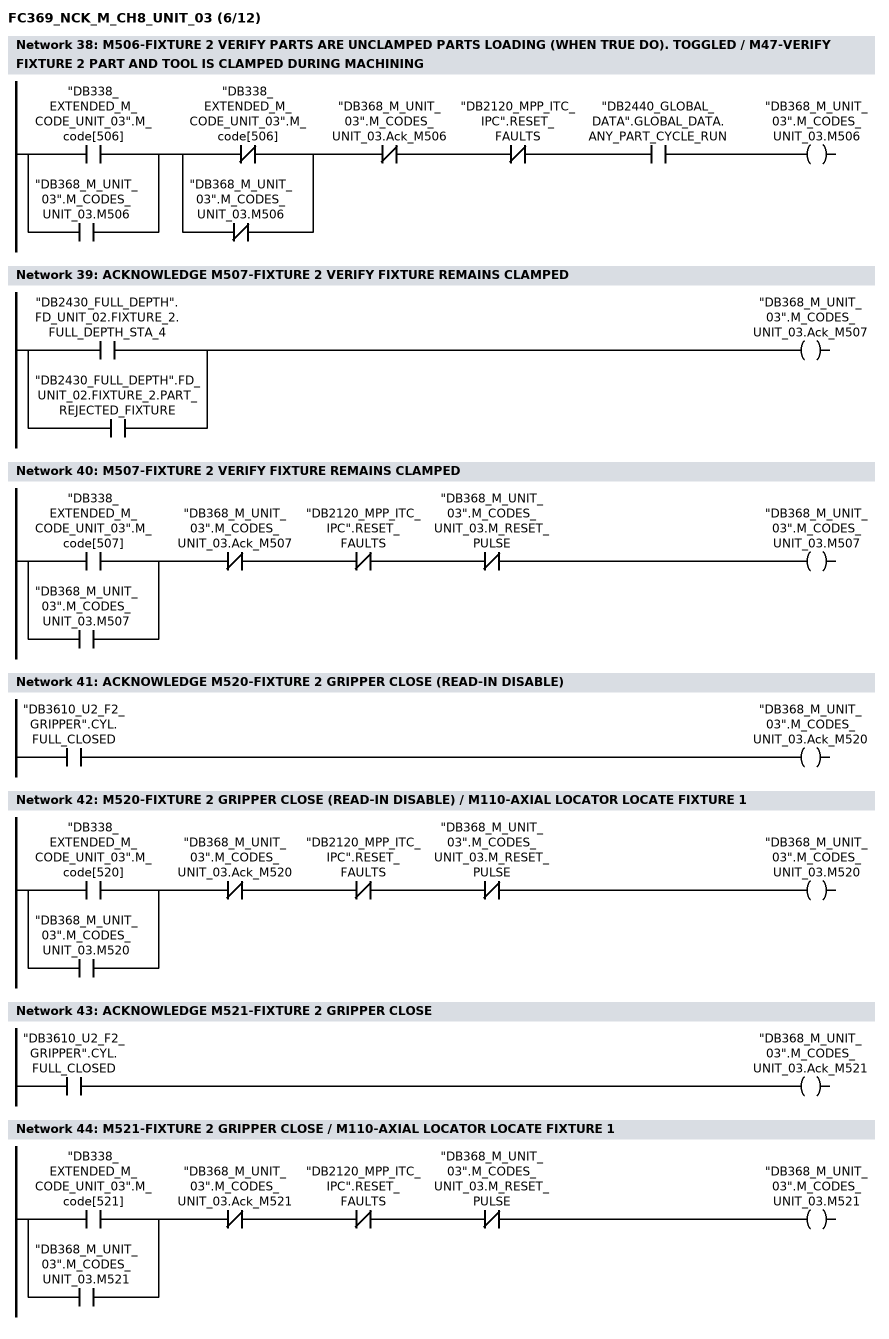
   RUNG wire#powerrail
      Contact( "DB338_EXTENDED_M_CODE_UNIT_03".M_code[506] )
      wire#w1
      I_Contact( "DB338_EXTENDED_M_CODE_UNIT_03".M_code[506] )
      wire#w2
      I_Contact( "DB368_M_UNIT_03".M_CODES_UNIT_03.Ack_M506 )
      I_Contact( "DB2120_MPP_ITC_IPC".RESET_FAULTS )
      Contact( "DB2440_GLOBAL_DATA".GLOBAL_DATA.ANY_PART_CYCLE_RUN )
      Coil( "DB368_M_UNIT_03".M_CODES_UNIT_03.M506 )
   END_RUNG
   RUNG wire#powerrail
      Contact( "DB368_M_UNIT_03".M_CODES_UNIT_03.M506 )
   END_RUNG wire#w1
   RUNG wire#w1
      I_Contact( "DB368_M_UNIT_03".M_CODES_UNIT_03.M506 )
   END_RUNG wire#w2
   // the same network as SCL:
   "DB368_M_UNIT_03".M_CODES_UNIT_03.M506 := ("DB338_EXTENDED_M_CODE_UNIT_03".M_code[506] OR "DB368_M_UNIT_03".M_CODES_UNIT_03.M506) AND (NOT "DB338_EXTENDED_M_CODE_UNIT_03".M_code[506] OR NOT "DB368_M_UNIT_03".M_CODES_UNIT_03.M506) AND NOT "DB368_M_UNIT_03".M_CODES_UNIT_03.Ack_M506 AND NOT "DB2120_MPP_ITC_IPC".RESET_FAULTS AND "DB2440_GLOBAL_DATA".GLOBAL_DATA.ANY_PART_CYCLE_RUN;
END_REGION

REGION Network 39: ACKNOWLEDGE M507-FIXTURE 2 VERIFY FIXTURE REMAINS CLAMPED
   RUNG wire#powerrail
      Contact( "DB2430_FULL_DEPTH".FD_UNIT_02.FIXTURE_2.FULL_DEPTH_STA_4 )
      wire#w1
      Coil( "DB368_M_UNIT_03".M_CODES_UNIT_03.Ack_M507 )
   END_RUNG
   RUNG wire#powerrail
      Contact( "DB2430_FULL_DEPTH".FD_UNIT_02.FIXTURE_2.PART_REJECTED_FIXTURE )
   END_RUNG wire#w1
   // the same network as SCL:
   "DB368_M_UNIT_03".M_CODES_UNIT_03.Ack_M507 := "DB2430_FULL_DEPTH".FD_UNIT_02.FIXTURE_2.FULL_DEPTH_STA_4 OR "DB2430_FULL_DEPTH".FD_UNIT_02.FIXTURE_2.PART_REJECTED_FIXTURE;
END_REGION

REGION Network 40: M507-FIXTURE 2 VERIFY FIXTURE REMAINS CLAMPED
   RUNG wire#powerrail
      Contact( "DB338_EXTENDED_M_CODE_UNIT_03".M_code[507] )
      wire#w1
      I_Contact( "DB368_M_UNIT_03".M_CODES_UNIT_03.Ack_M507 )
      I_Contact( "DB2120_MPP_ITC_IPC".RESET_FAULTS )
      I_Contact( "DB368_M_UNIT_03".M_CODES_UNIT_03.M_RESET_PULSE )
      Coil( "DB368_M_UNIT_03".M_CODES_UNIT_03.M507 )
   END_RUNG
   RUNG wire#powerrail
      Contact( "DB368_M_UNIT_03".M_CODES_UNIT_03.M507 )
   END_RUNG wire#w1
   // the same network as SCL:
   "DB368_M_UNIT_03".M_CODES_UNIT_03.M507 := ("DB338_EXTENDED_M_CODE_UNIT_03".M_code[507] OR "DB368_M_UNIT_03".M_CODES_UNIT_03.M507) AND NOT "DB368_M_UNIT_03".M_CODES_UNIT_03.Ack_M507 AND NOT "DB2120_MPP_ITC_IPC".RESET_FAULTS AND NOT "DB368_M_UNIT_03".M_CODES_UNIT_03.M_RESET_PULSE;
END_REGION

REGION Network 41: ACKNOWLEDGE M520-FIXTURE 2 GRIPPER CLOSE (READ-IN DISABLE)
   RUNG wire#powerrail
      Contact( "DB3610_U2_F2_GRIPPER".CYL.FULL_CLOSED )
      Coil( "DB368_M_UNIT_03".M_CODES_UNIT_03.Ack_M520 )
   END_RUNG
   // the same network as SCL:
   "DB368_M_UNIT_03".M_CODES_UNIT_03.Ack_M520 := "DB3610_U2_F2_GRIPPER".CYL.FULL_CLOSED;
END_REGION

REGION Network 42: M520-FIXTURE 2 GRIPPER CLOSE (READ-IN DISABLE) / M110-AXIAL LOCATOR LOCATE FIXTURE 1
   RUNG wire#powerrail
      Contact( "DB338_EXTENDED_M_CODE_UNIT_03".M_code[520] )
      wire#w1
      I_Contact( "DB368_M_UNIT_03".M_CODES_UNIT_03.Ack_M520 )
      I_Contact( "DB2120_MPP_ITC_IPC".RESET_FAULTS )
      I_Contact( "DB368_M_UNIT_03".M_CODES_UNIT_03.M_RESET_PULSE )
      Coil( "DB368_M_UNIT_03".M_CODES_UNIT_03.M520 )
   END_RUNG
   RUNG wire#powerrail
      Contact( "DB368_M_UNIT_03".M_CODES_UNIT_03.M520 )
   END_RUNG wire#w1
   // the same network as SCL:
   "DB368_M_UNIT_03".M_CODES_UNIT_03.M520 := ("DB338_EXTENDED_M_CODE_UNIT_03".M_code[520] OR "DB368_M_UNIT_03".M_CODES_UNIT_03.M520) AND NOT "DB368_M_UNIT_03".M_CODES_UNIT_03.Ack_M520 AND NOT "DB2120_MPP_ITC_IPC".RESET_FAULTS AND NOT "DB368_M_UNIT_03".M_CODES_UNIT_03.M_RESET_PULSE;
END_REGION

REGION Network 43: ACKNOWLEDGE M521-FIXTURE 2 GRIPPER CLOSE
   RUNG wire#powerrail
      Contact( "DB3610_U2_F2_GRIPPER".CYL.FULL_CLOSED )
      Coil( "DB368_M_UNIT_03".M_CODES_UNIT_03.Ack_M521 )
   END_RUNG
   // the same network as SCL:
   "DB368_M_UNIT_03".M_CODES_UNIT_03.Ack_M521 := "DB3610_U2_F2_GRIPPER".CYL.FULL_CLOSED;
END_REGION

REGION Network 44: M521-FIXTURE 2 GRIPPER CLOSE / M110-AXIAL LOCATOR LOCATE FIXTURE 1
   RUNG wire#powerrail
      Contact( "DB338_EXTENDED_M_CODE_UNIT_03".M_code[521] )
      wire#w1
      I_Contact( "DB368_M_UNIT_03".M_CODES_UNIT_03.Ack_M521 )
      I_Contact( "DB2120_MPP_ITC_IPC".RESET_FAULTS )
      I_Contact( "DB368_M_UNIT_03".M_CODES_UNIT_03.M_RESET_PULSE )
      Coil( "DB368_M_UNIT_03".M_CODES_UNIT_03.M521 )
   END_RUNG
   RUNG wire#powerrail
      Contact( "DB368_M_UNIT_03".M_CODES_UNIT_03.M521 )
   END_RUNG wire#w1
   // the same network as SCL:
   "DB368_M_UNIT_03".M_CODES_UNIT_03.M521 := ("DB338_EXTENDED_M_CODE_UNIT_03".M_code[521] OR "DB368_M_UNIT_03".M_CODES_UNIT_03.M521) AND NOT "DB368_M_UNIT_03".M_CODES_UNIT_03.Ack_M521 AND NOT "DB2120_MPP_ITC_IPC".RESET_FAULTS AND NOT "DB368_M_UNIT_03".M_CODES_UNIT_03.M_RESET_PULSE;
END_REGION

REGION Network 45: ACKNOWLEDGE M522-FIXTURE 2 GRIPPER RETURN (READ-IN DISABLE) / ACKNOWLEDGE M111-AXIAL LOCATOR RETURN FIXTURE 1
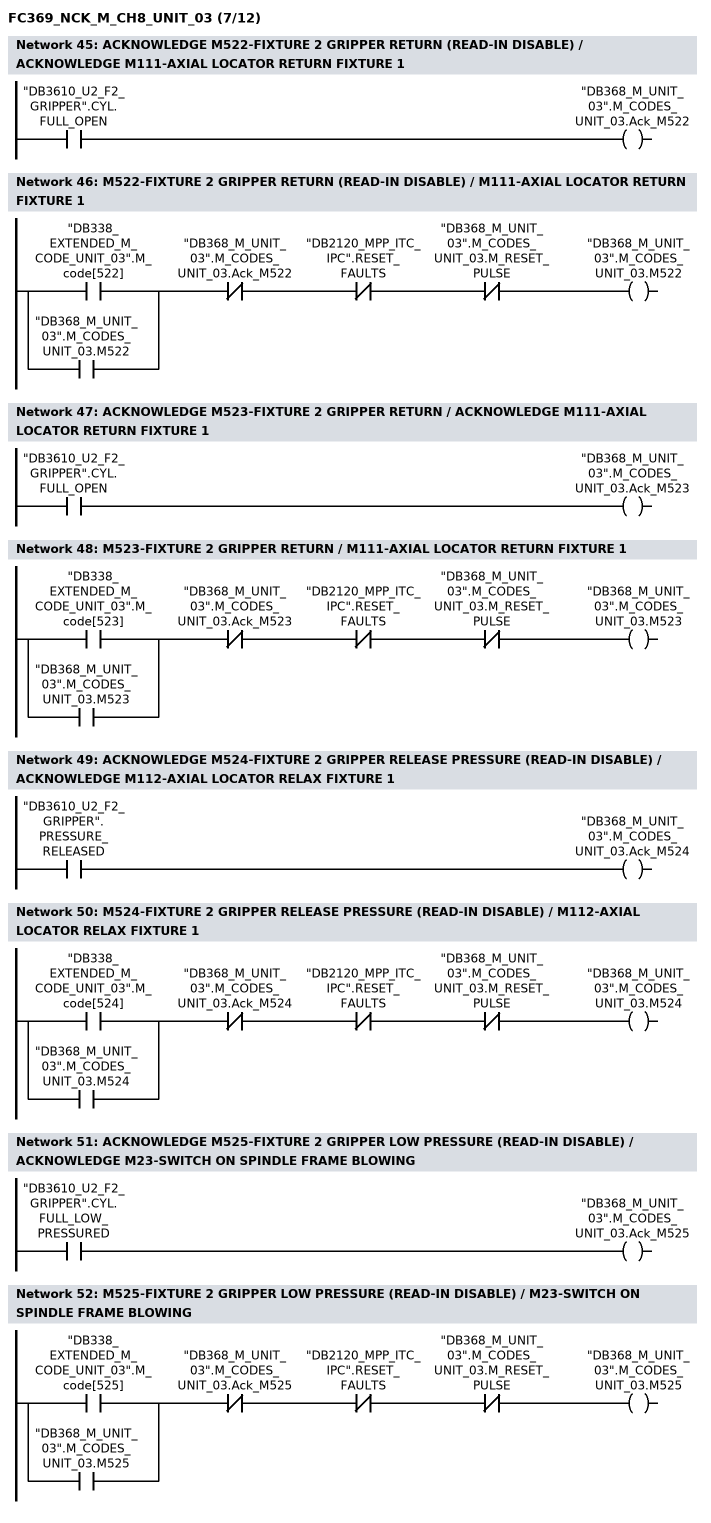
   RUNG wire#powerrail
      Contact( "DB3610_U2_F2_GRIPPER".CYL.FULL_OPEN )
      Coil( "DB368_M_UNIT_03".M_CODES_UNIT_03.Ack_M522 )
   END_RUNG
   // the same network as SCL:
   "DB368_M_UNIT_03".M_CODES_UNIT_03.Ack_M522 := "DB3610_U2_F2_GRIPPER".CYL.FULL_OPEN;
END_REGION

REGION Network 46: M522-FIXTURE 2 GRIPPER RETURN (READ-IN DISABLE) / M111-AXIAL LOCATOR RETURN FIXTURE 1
   RUNG wire#powerrail
      Contact( "DB338_EXTENDED_M_CODE_UNIT_03".M_code[522] )
      wire#w1
      I_Contact( "DB368_M_UNIT_03".M_CODES_UNIT_03.Ack_M522 )
      I_Contact( "DB2120_MPP_ITC_IPC".RESET_FAULTS )
      I_Contact( "DB368_M_UNIT_03".M_CODES_UNIT_03.M_RESET_PULSE )
      Coil( "DB368_M_UNIT_03".M_CODES_UNIT_03.M522 )
   END_RUNG
   RUNG wire#powerrail
      Contact( "DB368_M_UNIT_03".M_CODES_UNIT_03.M522 )
   END_RUNG wire#w1
   // the same network as SCL:
   "DB368_M_UNIT_03".M_CODES_UNIT_03.M522 := ("DB338_EXTENDED_M_CODE_UNIT_03".M_code[522] OR "DB368_M_UNIT_03".M_CODES_UNIT_03.M522) AND NOT "DB368_M_UNIT_03".M_CODES_UNIT_03.Ack_M522 AND NOT "DB2120_MPP_ITC_IPC".RESET_FAULTS AND NOT "DB368_M_UNIT_03".M_CODES_UNIT_03.M_RESET_PULSE;
END_REGION

REGION Network 47: ACKNOWLEDGE M523-FIXTURE 2 GRIPPER RETURN / ACKNOWLEDGE M111-AXIAL LOCATOR RETURN FIXTURE 1
   RUNG wire#powerrail
      Contact( "DB3610_U2_F2_GRIPPER".CYL.FULL_OPEN )
      Coil( "DB368_M_UNIT_03".M_CODES_UNIT_03.Ack_M523 )
   END_RUNG
   // the same network as SCL:
   "DB368_M_UNIT_03".M_CODES_UNIT_03.Ack_M523 := "DB3610_U2_F2_GRIPPER".CYL.FULL_OPEN;
END_REGION

REGION Network 48: M523-FIXTURE 2 GRIPPER RETURN / M111-AXIAL LOCATOR RETURN FIXTURE 1
   RUNG wire#powerrail
      Contact( "DB338_EXTENDED_M_CODE_UNIT_03".M_code[523] )
      wire#w1
      I_Contact( "DB368_M_UNIT_03".M_CODES_UNIT_03.Ack_M523 )
      I_Contact( "DB2120_MPP_ITC_IPC".RESET_FAULTS )
      I_Contact( "DB368_M_UNIT_03".M_CODES_UNIT_03.M_RESET_PULSE )
      Coil( "DB368_M_UNIT_03".M_CODES_UNIT_03.M523 )
   END_RUNG
   RUNG wire#powerrail
      Contact( "DB368_M_UNIT_03".M_CODES_UNIT_03.M523 )
   END_RUNG wire#w1
   // the same network as SCL:
   "DB368_M_UNIT_03".M_CODES_UNIT_03.M523 := ("DB338_EXTENDED_M_CODE_UNIT_03".M_code[523] OR "DB368_M_UNIT_03".M_CODES_UNIT_03.M523) AND NOT "DB368_M_UNIT_03".M_CODES_UNIT_03.Ack_M523 AND NOT "DB2120_MPP_ITC_IPC".RESET_FAULTS AND NOT "DB368_M_UNIT_03".M_CODES_UNIT_03.M_RESET_PULSE;
END_REGION

REGION Network 49: ACKNOWLEDGE M524-FIXTURE 2 GRIPPER RELEASE PRESSURE (READ-IN DISABLE) / ACKNOWLEDGE M112-AXIAL LOCATOR RELAX FIXTURE 1
   RUNG wire#powerrail
      Contact( "DB3610_U2_F2_GRIPPER".PRESSURE_RELEASED )
      Coil( "DB368_M_UNIT_03".M_CODES_UNIT_03.Ack_M524 )
   END_RUNG
   // the same network as SCL:
   "DB368_M_UNIT_03".M_CODES_UNIT_03.Ack_M524 := "DB3610_U2_F2_GRIPPER".PRESSURE_RELEASED;
END_REGION

REGION Network 50: M524-FIXTURE 2 GRIPPER RELEASE PRESSURE (READ-IN DISABLE) / M112-AXIAL LOCATOR RELAX FIXTURE 1
   RUNG wire#powerrail
      Contact( "DB338_EXTENDED_M_CODE_UNIT_03".M_code[524] )
      wire#w1
      I_Contact( "DB368_M_UNIT_03".M_CODES_UNIT_03.Ack_M524 )
      I_Contact( "DB2120_MPP_ITC_IPC".RESET_FAULTS )
      I_Contact( "DB368_M_UNIT_03".M_CODES_UNIT_03.M_RESET_PULSE )
      Coil( "DB368_M_UNIT_03".M_CODES_UNIT_03.M524 )
   END_RUNG
   RUNG wire#powerrail
      Contact( "DB368_M_UNIT_03".M_CODES_UNIT_03.M524 )
   END_RUNG wire#w1
   // the same network as SCL:
   "DB368_M_UNIT_03".M_CODES_UNIT_03.M524 := ("DB338_EXTENDED_M_CODE_UNIT_03".M_code[524] OR "DB368_M_UNIT_03".M_CODES_UNIT_03.M524) AND NOT "DB368_M_UNIT_03".M_CODES_UNIT_03.Ack_M524 AND NOT "DB2120_MPP_ITC_IPC".RESET_FAULTS AND NOT "DB368_M_UNIT_03".M_CODES_UNIT_03.M_RESET_PULSE;
END_REGION

REGION Network 51: ACKNOWLEDGE M525-FIXTURE 2 GRIPPER LOW PRESSURE (READ-IN DISABLE) / ACKNOWLEDGE M23-SWITCH ON SPINDLE FRAME BLOWING
   RUNG wire#powerrail
      Contact( "DB3610_U2_F2_GRIPPER".CYL.FULL_LOW_PRESSURED )
      Coil( "DB368_M_UNIT_03".M_CODES_UNIT_03.Ack_M525 )
   END_RUNG
   // the same network as SCL:
   "DB368_M_UNIT_03".M_CODES_UNIT_03.Ack_M525 := "DB3610_U2_F2_GRIPPER".CYL.FULL_LOW_PRESSURED;
END_REGION

REGION Network 52: M525-FIXTURE 2 GRIPPER LOW PRESSURE (READ-IN DISABLE) / M23-SWITCH ON SPINDLE FRAME BLOWING
   RUNG wire#powerrail
      Contact( "DB338_EXTENDED_M_CODE_UNIT_03".M_code[525] )
      wire#w1
      I_Contact( "DB368_M_UNIT_03".M_CODES_UNIT_03.Ack_M525 )
      I_Contact( "DB2120_MPP_ITC_IPC".RESET_FAULTS )
      I_Contact( "DB368_M_UNIT_03".M_CODES_UNIT_03.M_RESET_PULSE )
      Coil( "DB368_M_UNIT_03".M_CODES_UNIT_03.M525 )
   END_RUNG
   RUNG wire#powerrail
      Contact( "DB368_M_UNIT_03".M_CODES_UNIT_03.M525 )
   END_RUNG wire#w1
   // the same network as SCL:
   "DB368_M_UNIT_03".M_CODES_UNIT_03.M525 := ("DB338_EXTENDED_M_CODE_UNIT_03".M_code[525] OR "DB368_M_UNIT_03".M_CODES_UNIT_03.M525) AND NOT "DB368_M_UNIT_03".M_CODES_UNIT_03.Ack_M525 AND NOT "DB2120_MPP_ITC_IPC".RESET_FAULTS AND NOT "DB368_M_UNIT_03".M_CODES_UNIT_03.M_RESET_PULSE;
END_REGION

REGION Network 53: ACKNOWLEDGE M600-FIXTURE 3 CLAMP SEQUENCE (READ-IN DISABLE) / ACKNOWLEDGE M100-CLAMP SEQUENCE FIXTURE 1
   // NOTE: WHEN THERE IS NOT INDEXING TABLE AVAILABLE IN THE MACHINE DELETE 
   // DB2171.DBX5.0 AND DB2171.DBX2.0
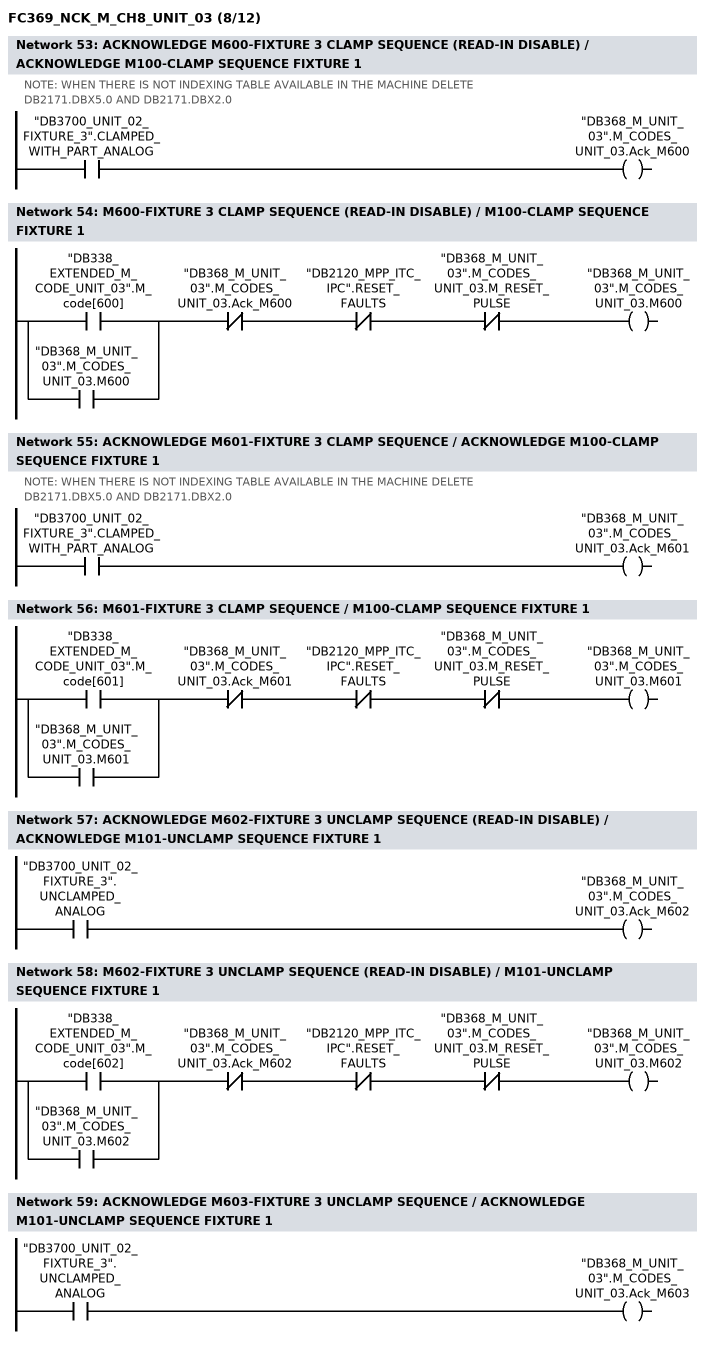
   RUNG wire#powerrail
      Contact( "DB3700_UNIT_02_FIXTURE_3".CLAMPED_WITH_PART_ANALOG )
      Coil( "DB368_M_UNIT_03".M_CODES_UNIT_03.Ack_M600 )
   END_RUNG
   // the same network as SCL:
   "DB368_M_UNIT_03".M_CODES_UNIT_03.Ack_M600 := "DB3700_UNIT_02_FIXTURE_3".CLAMPED_WITH_PART_ANALOG;
END_REGION

REGION Network 54: M600-FIXTURE 3 CLAMP SEQUENCE (READ-IN DISABLE) / M100-CLAMP SEQUENCE FIXTURE 1
   RUNG wire#powerrail
      Contact( "DB338_EXTENDED_M_CODE_UNIT_03".M_code[600] )
      wire#w1
      I_Contact( "DB368_M_UNIT_03".M_CODES_UNIT_03.Ack_M600 )
      I_Contact( "DB2120_MPP_ITC_IPC".RESET_FAULTS )
      I_Contact( "DB368_M_UNIT_03".M_CODES_UNIT_03.M_RESET_PULSE )
      Coil( "DB368_M_UNIT_03".M_CODES_UNIT_03.M600 )
   END_RUNG
   RUNG wire#powerrail
      Contact( "DB368_M_UNIT_03".M_CODES_UNIT_03.M600 )
   END_RUNG wire#w1
   // the same network as SCL:
   "DB368_M_UNIT_03".M_CODES_UNIT_03.M600 := ("DB338_EXTENDED_M_CODE_UNIT_03".M_code[600] OR "DB368_M_UNIT_03".M_CODES_UNIT_03.M600) AND NOT "DB368_M_UNIT_03".M_CODES_UNIT_03.Ack_M600 AND NOT "DB2120_MPP_ITC_IPC".RESET_FAULTS AND NOT "DB368_M_UNIT_03".M_CODES_UNIT_03.M_RESET_PULSE;
END_REGION

REGION Network 55: ACKNOWLEDGE M601-FIXTURE 3 CLAMP SEQUENCE / ACKNOWLEDGE M100-CLAMP SEQUENCE FIXTURE 1
   // NOTE: WHEN THERE IS NOT INDEXING TABLE AVAILABLE IN THE MACHINE DELETE 
   // DB2171.DBX5.0 AND DB2171.DBX2.0
   RUNG wire#powerrail
      Contact( "DB3700_UNIT_02_FIXTURE_3".CLAMPED_WITH_PART_ANALOG )
      Coil( "DB368_M_UNIT_03".M_CODES_UNIT_03.Ack_M601 )
   END_RUNG
   // the same network as SCL:
   "DB368_M_UNIT_03".M_CODES_UNIT_03.Ack_M601 := "DB3700_UNIT_02_FIXTURE_3".CLAMPED_WITH_PART_ANALOG;
END_REGION

REGION Network 56: M601-FIXTURE 3 CLAMP SEQUENCE / M100-CLAMP SEQUENCE FIXTURE 1
   RUNG wire#powerrail
      Contact( "DB338_EXTENDED_M_CODE_UNIT_03".M_code[601] )
      wire#w1
      I_Contact( "DB368_M_UNIT_03".M_CODES_UNIT_03.Ack_M601 )
      I_Contact( "DB2120_MPP_ITC_IPC".RESET_FAULTS )
      I_Contact( "DB368_M_UNIT_03".M_CODES_UNIT_03.M_RESET_PULSE )
      Coil( "DB368_M_UNIT_03".M_CODES_UNIT_03.M601 )
   END_RUNG
   RUNG wire#powerrail
      Contact( "DB368_M_UNIT_03".M_CODES_UNIT_03.M601 )
   END_RUNG wire#w1
   // the same network as SCL:
   "DB368_M_UNIT_03".M_CODES_UNIT_03.M601 := ("DB338_EXTENDED_M_CODE_UNIT_03".M_code[601] OR "DB368_M_UNIT_03".M_CODES_UNIT_03.M601) AND NOT "DB368_M_UNIT_03".M_CODES_UNIT_03.Ack_M601 AND NOT "DB2120_MPP_ITC_IPC".RESET_FAULTS AND NOT "DB368_M_UNIT_03".M_CODES_UNIT_03.M_RESET_PULSE;
END_REGION

REGION Network 57: ACKNOWLEDGE M602-FIXTURE 3 UNCLAMP SEQUENCE (READ-IN DISABLE) / ACKNOWLEDGE M101-UNCLAMP SEQUENCE FIXTURE 1
   RUNG wire#powerrail
      Contact( "DB3700_UNIT_02_FIXTURE_3".UNCLAMPED_ANALOG )
      Coil( "DB368_M_UNIT_03".M_CODES_UNIT_03.Ack_M602 )
   END_RUNG
   // the same network as SCL:
   "DB368_M_UNIT_03".M_CODES_UNIT_03.Ack_M602 := "DB3700_UNIT_02_FIXTURE_3".UNCLAMPED_ANALOG;
END_REGION

REGION Network 58: M602-FIXTURE 3 UNCLAMP SEQUENCE (READ-IN DISABLE) / M101-UNCLAMP SEQUENCE FIXTURE 1
   RUNG wire#powerrail
      Contact( "DB338_EXTENDED_M_CODE_UNIT_03".M_code[602] )
      wire#w1
      I_Contact( "DB368_M_UNIT_03".M_CODES_UNIT_03.Ack_M602 )
      I_Contact( "DB2120_MPP_ITC_IPC".RESET_FAULTS )
      I_Contact( "DB368_M_UNIT_03".M_CODES_UNIT_03.M_RESET_PULSE )
      Coil( "DB368_M_UNIT_03".M_CODES_UNIT_03.M602 )
   END_RUNG
   RUNG wire#powerrail
      Contact( "DB368_M_UNIT_03".M_CODES_UNIT_03.M602 )
   END_RUNG wire#w1
   // the same network as SCL:
   "DB368_M_UNIT_03".M_CODES_UNIT_03.M602 := ("DB338_EXTENDED_M_CODE_UNIT_03".M_code[602] OR "DB368_M_UNIT_03".M_CODES_UNIT_03.M602) AND NOT "DB368_M_UNIT_03".M_CODES_UNIT_03.Ack_M602 AND NOT "DB2120_MPP_ITC_IPC".RESET_FAULTS AND NOT "DB368_M_UNIT_03".M_CODES_UNIT_03.M_RESET_PULSE;
END_REGION

REGION Network 59: ACKNOWLEDGE M603-FIXTURE 3 UNCLAMP SEQUENCE / ACKNOWLEDGE M101-UNCLAMP SEQUENCE FIXTURE 1
   RUNG wire#powerrail
      Contact( "DB3700_UNIT_02_FIXTURE_3".UNCLAMPED_ANALOG )
      Coil( "DB368_M_UNIT_03".M_CODES_UNIT_03.Ack_M603 )
   END_RUNG
   // the same network as SCL:
   "DB368_M_UNIT_03".M_CODES_UNIT_03.Ack_M603 := "DB3700_UNIT_02_FIXTURE_3".UNCLAMPED_ANALOG;
END_REGION

REGION Network 60: M603-FIXTURE 3 UNCLAMP SEQUENCE / M101-UNCLAMP SEQUENCE FIXTURE 1
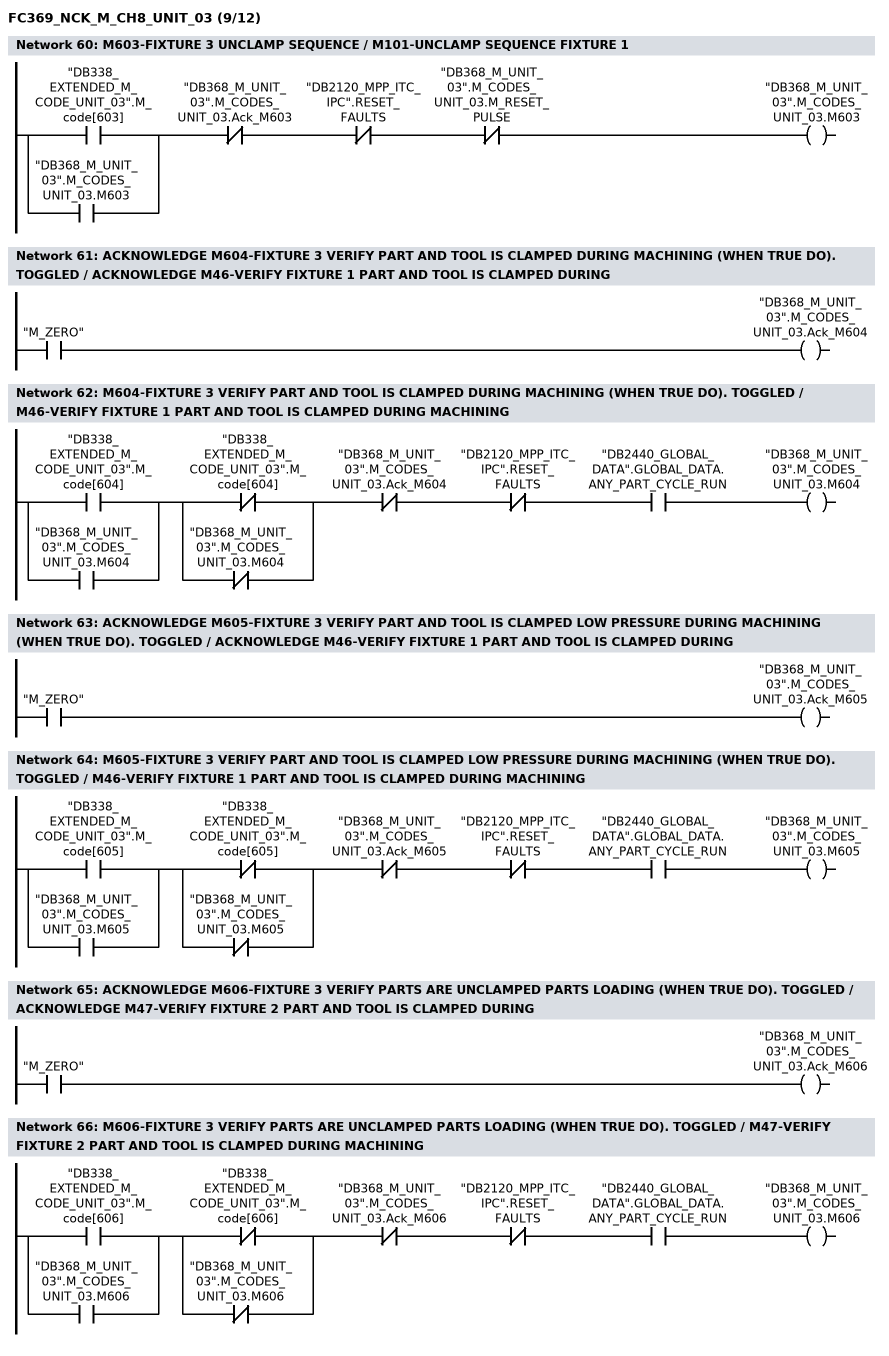
   RUNG wire#powerrail
      Contact( "DB338_EXTENDED_M_CODE_UNIT_03".M_code[603] )
      wire#w1
      I_Contact( "DB368_M_UNIT_03".M_CODES_UNIT_03.Ack_M603 )
      I_Contact( "DB2120_MPP_ITC_IPC".RESET_FAULTS )
      I_Contact( "DB368_M_UNIT_03".M_CODES_UNIT_03.M_RESET_PULSE )
      Coil( "DB368_M_UNIT_03".M_CODES_UNIT_03.M603 )
   END_RUNG
   RUNG wire#powerrail
      Contact( "DB368_M_UNIT_03".M_CODES_UNIT_03.M603 )
   END_RUNG wire#w1
   // the same network as SCL:
   "DB368_M_UNIT_03".M_CODES_UNIT_03.M603 := ("DB338_EXTENDED_M_CODE_UNIT_03".M_code[603] OR "DB368_M_UNIT_03".M_CODES_UNIT_03.M603) AND NOT "DB368_M_UNIT_03".M_CODES_UNIT_03.Ack_M603 AND NOT "DB2120_MPP_ITC_IPC".RESET_FAULTS AND NOT "DB368_M_UNIT_03".M_CODES_UNIT_03.M_RESET_PULSE;
END_REGION

REGION Network 61: ACKNOWLEDGE M604-FIXTURE 3 VERIFY PART AND TOOL IS CLAMPED DURING MACHINING (WHEN TRUE DO). TOGGLED / ACKNOWLEDGE M46-VERIFY FIXTURE 1 PART AND TOOL IS CLAMPED DURING
   RUNG wire#powerrail
      Contact( "M_ZERO" )
      Coil( "DB368_M_UNIT_03".M_CODES_UNIT_03.Ack_M604 )
   END_RUNG
   // the same network as SCL:
   "DB368_M_UNIT_03".M_CODES_UNIT_03.Ack_M604 := "M_ZERO";
END_REGION

REGION Network 62: M604-FIXTURE 3 VERIFY PART AND TOOL IS CLAMPED DURING MACHINING (WHEN TRUE DO). TOGGLED / M46-VERIFY FIXTURE 1 PART AND TOOL IS CLAMPED DURING MACHINING
   RUNG wire#powerrail
      Contact( "DB338_EXTENDED_M_CODE_UNIT_03".M_code[604] )
      wire#w1
      I_Contact( "DB338_EXTENDED_M_CODE_UNIT_03".M_code[604] )
      wire#w2
      I_Contact( "DB368_M_UNIT_03".M_CODES_UNIT_03.Ack_M604 )
      I_Contact( "DB2120_MPP_ITC_IPC".RESET_FAULTS )
      Contact( "DB2440_GLOBAL_DATA".GLOBAL_DATA.ANY_PART_CYCLE_RUN )
      Coil( "DB368_M_UNIT_03".M_CODES_UNIT_03.M604 )
   END_RUNG
   RUNG wire#powerrail
      Contact( "DB368_M_UNIT_03".M_CODES_UNIT_03.M604 )
   END_RUNG wire#w1
   RUNG wire#w1
      I_Contact( "DB368_M_UNIT_03".M_CODES_UNIT_03.M604 )
   END_RUNG wire#w2
   // the same network as SCL:
   "DB368_M_UNIT_03".M_CODES_UNIT_03.M604 := ("DB338_EXTENDED_M_CODE_UNIT_03".M_code[604] OR "DB368_M_UNIT_03".M_CODES_UNIT_03.M604) AND (NOT "DB338_EXTENDED_M_CODE_UNIT_03".M_code[604] OR NOT "DB368_M_UNIT_03".M_CODES_UNIT_03.M604) AND NOT "DB368_M_UNIT_03".M_CODES_UNIT_03.Ack_M604 AND NOT "DB2120_MPP_ITC_IPC".RESET_FAULTS AND "DB2440_GLOBAL_DATA".GLOBAL_DATA.ANY_PART_CYCLE_RUN;
END_REGION

REGION Network 63: ACKNOWLEDGE M605-FIXTURE 3 VERIFY PART AND TOOL IS CLAMPED LOW PRESSURE DURING MACHINING (WHEN TRUE DO). TOGGLED / ACKNOWLEDGE M46-VERIFY FIXTURE 1 PART AND TOOL IS CLAMPED DURING
   RUNG wire#powerrail
      Contact( "M_ZERO" )
      Coil( "DB368_M_UNIT_03".M_CODES_UNIT_03.Ack_M605 )
   END_RUNG
   // the same network as SCL:
   "DB368_M_UNIT_03".M_CODES_UNIT_03.Ack_M605 := "M_ZERO";
END_REGION

REGION Network 64: M605-FIXTURE 3 VERIFY PART AND TOOL IS CLAMPED LOW PRESSURE DURING MACHINING (WHEN TRUE DO). TOGGLED / M46-VERIFY FIXTURE 1 PART AND TOOL IS CLAMPED DURING MACHINING
   RUNG wire#powerrail
      Contact( "DB338_EXTENDED_M_CODE_UNIT_03".M_code[605] )
      wire#w1
      I_Contact( "DB338_EXTENDED_M_CODE_UNIT_03".M_code[605] )
      wire#w2
      I_Contact( "DB368_M_UNIT_03".M_CODES_UNIT_03.Ack_M605 )
      I_Contact( "DB2120_MPP_ITC_IPC".RESET_FAULTS )
      Contact( "DB2440_GLOBAL_DATA".GLOBAL_DATA.ANY_PART_CYCLE_RUN )
      Coil( "DB368_M_UNIT_03".M_CODES_UNIT_03.M605 )
   END_RUNG
   RUNG wire#powerrail
      Contact( "DB368_M_UNIT_03".M_CODES_UNIT_03.M605 )
   END_RUNG wire#w1
   RUNG wire#w1
      I_Contact( "DB368_M_UNIT_03".M_CODES_UNIT_03.M605 )
   END_RUNG wire#w2
   // the same network as SCL:
   "DB368_M_UNIT_03".M_CODES_UNIT_03.M605 := ("DB338_EXTENDED_M_CODE_UNIT_03".M_code[605] OR "DB368_M_UNIT_03".M_CODES_UNIT_03.M605) AND (NOT "DB338_EXTENDED_M_CODE_UNIT_03".M_code[605] OR NOT "DB368_M_UNIT_03".M_CODES_UNIT_03.M605) AND NOT "DB368_M_UNIT_03".M_CODES_UNIT_03.Ack_M605 AND NOT "DB2120_MPP_ITC_IPC".RESET_FAULTS AND "DB2440_GLOBAL_DATA".GLOBAL_DATA.ANY_PART_CYCLE_RUN;
END_REGION

REGION Network 65: ACKNOWLEDGE M606-FIXTURE 3 VERIFY PARTS ARE UNCLAMPED PARTS LOADING (WHEN TRUE DO). TOGGLED / ACKNOWLEDGE M47-VERIFY FIXTURE 2 PART AND TOOL IS CLAMPED DURING
   RUNG wire#powerrail
      Contact( "M_ZERO" )
      Coil( "DB368_M_UNIT_03".M_CODES_UNIT_03.Ack_M606 )
   END_RUNG
   // the same network as SCL:
   "DB368_M_UNIT_03".M_CODES_UNIT_03.Ack_M606 := "M_ZERO";
END_REGION

REGION Network 66: M606-FIXTURE 3 VERIFY PARTS ARE UNCLAMPED PARTS LOADING (WHEN TRUE DO). TOGGLED / M47-VERIFY FIXTURE 2 PART AND TOOL IS CLAMPED DURING MACHINING
   RUNG wire#powerrail
      Contact( "DB338_EXTENDED_M_CODE_UNIT_03".M_code[606] )
      wire#w1
      I_Contact( "DB338_EXTENDED_M_CODE_UNIT_03".M_code[606] )
      wire#w2
      I_Contact( "DB368_M_UNIT_03".M_CODES_UNIT_03.Ack_M606 )
      I_Contact( "DB2120_MPP_ITC_IPC".RESET_FAULTS )
      Contact( "DB2440_GLOBAL_DATA".GLOBAL_DATA.ANY_PART_CYCLE_RUN )
      Coil( "DB368_M_UNIT_03".M_CODES_UNIT_03.M606 )
   END_RUNG
   RUNG wire#powerrail
      Contact( "DB368_M_UNIT_03".M_CODES_UNIT_03.M606 )
   END_RUNG wire#w1
   RUNG wire#w1
      I_Contact( "DB368_M_UNIT_03".M_CODES_UNIT_03.M606 )
   END_RUNG wire#w2
   // the same network as SCL:
   "DB368_M_UNIT_03".M_CODES_UNIT_03.M606 := ("DB338_EXTENDED_M_CODE_UNIT_03".M_code[606] OR "DB368_M_UNIT_03".M_CODES_UNIT_03.M606) AND (NOT "DB338_EXTENDED_M_CODE_UNIT_03".M_code[606] OR NOT "DB368_M_UNIT_03".M_CODES_UNIT_03.M606) AND NOT "DB368_M_UNIT_03".M_CODES_UNIT_03.Ack_M606 AND NOT "DB2120_MPP_ITC_IPC".RESET_FAULTS AND "DB2440_GLOBAL_DATA".GLOBAL_DATA.ANY_PART_CYCLE_RUN;
END_REGION

REGION Network 67: ACKNOWLEDGE M607-FIXTURE 3 VERIFY FIXTURE REMAINS CLAMPED
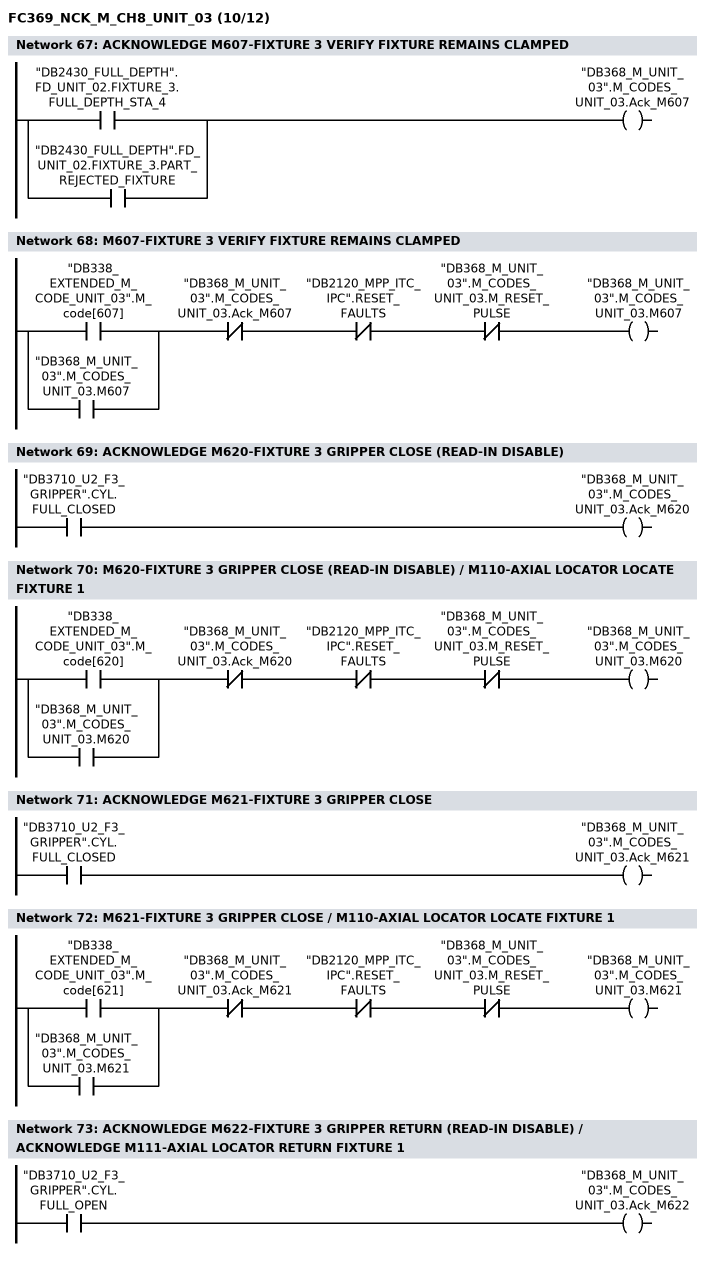
   RUNG wire#powerrail
      Contact( "DB2430_FULL_DEPTH".FD_UNIT_02.FIXTURE_3.FULL_DEPTH_STA_4 )
      wire#w1
      Coil( "DB368_M_UNIT_03".M_CODES_UNIT_03.Ack_M607 )
   END_RUNG
   RUNG wire#powerrail
      Contact( "DB2430_FULL_DEPTH".FD_UNIT_02.FIXTURE_3.PART_REJECTED_FIXTURE )
   END_RUNG wire#w1
   // the same network as SCL:
   "DB368_M_UNIT_03".M_CODES_UNIT_03.Ack_M607 := "DB2430_FULL_DEPTH".FD_UNIT_02.FIXTURE_3.FULL_DEPTH_STA_4 OR "DB2430_FULL_DEPTH".FD_UNIT_02.FIXTURE_3.PART_REJECTED_FIXTURE;
END_REGION

REGION Network 68: M607-FIXTURE 3 VERIFY FIXTURE REMAINS CLAMPED
   RUNG wire#powerrail
      Contact( "DB338_EXTENDED_M_CODE_UNIT_03".M_code[607] )
      wire#w1
      I_Contact( "DB368_M_UNIT_03".M_CODES_UNIT_03.Ack_M607 )
      I_Contact( "DB2120_MPP_ITC_IPC".RESET_FAULTS )
      I_Contact( "DB368_M_UNIT_03".M_CODES_UNIT_03.M_RESET_PULSE )
      Coil( "DB368_M_UNIT_03".M_CODES_UNIT_03.M607 )
   END_RUNG
   RUNG wire#powerrail
      Contact( "DB368_M_UNIT_03".M_CODES_UNIT_03.M607 )
   END_RUNG wire#w1
   // the same network as SCL:
   "DB368_M_UNIT_03".M_CODES_UNIT_03.M607 := ("DB338_EXTENDED_M_CODE_UNIT_03".M_code[607] OR "DB368_M_UNIT_03".M_CODES_UNIT_03.M607) AND NOT "DB368_M_UNIT_03".M_CODES_UNIT_03.Ack_M607 AND NOT "DB2120_MPP_ITC_IPC".RESET_FAULTS AND NOT "DB368_M_UNIT_03".M_CODES_UNIT_03.M_RESET_PULSE;
END_REGION

REGION Network 69: ACKNOWLEDGE M620-FIXTURE 3 GRIPPER CLOSE (READ-IN DISABLE)
   RUNG wire#powerrail
      Contact( "DB3710_U2_F3_GRIPPER".CYL.FULL_CLOSED )
      Coil( "DB368_M_UNIT_03".M_CODES_UNIT_03.Ack_M620 )
   END_RUNG
   // the same network as SCL:
   "DB368_M_UNIT_03".M_CODES_UNIT_03.Ack_M620 := "DB3710_U2_F3_GRIPPER".CYL.FULL_CLOSED;
END_REGION

REGION Network 70: M620-FIXTURE 3 GRIPPER CLOSE (READ-IN DISABLE) / M110-AXIAL LOCATOR LOCATE FIXTURE 1
   RUNG wire#powerrail
      Contact( "DB338_EXTENDED_M_CODE_UNIT_03".M_code[620] )
      wire#w1
      I_Contact( "DB368_M_UNIT_03".M_CODES_UNIT_03.Ack_M620 )
      I_Contact( "DB2120_MPP_ITC_IPC".RESET_FAULTS )
      I_Contact( "DB368_M_UNIT_03".M_CODES_UNIT_03.M_RESET_PULSE )
      Coil( "DB368_M_UNIT_03".M_CODES_UNIT_03.M620 )
   END_RUNG
   RUNG wire#powerrail
      Contact( "DB368_M_UNIT_03".M_CODES_UNIT_03.M620 )
   END_RUNG wire#w1
   // the same network as SCL:
   "DB368_M_UNIT_03".M_CODES_UNIT_03.M620 := ("DB338_EXTENDED_M_CODE_UNIT_03".M_code[620] OR "DB368_M_UNIT_03".M_CODES_UNIT_03.M620) AND NOT "DB368_M_UNIT_03".M_CODES_UNIT_03.Ack_M620 AND NOT "DB2120_MPP_ITC_IPC".RESET_FAULTS AND NOT "DB368_M_UNIT_03".M_CODES_UNIT_03.M_RESET_PULSE;
END_REGION

REGION Network 71: ACKNOWLEDGE M621-FIXTURE 3 GRIPPER CLOSE
   RUNG wire#powerrail
      Contact( "DB3710_U2_F3_GRIPPER".CYL.FULL_CLOSED )
      Coil( "DB368_M_UNIT_03".M_CODES_UNIT_03.Ack_M621 )
   END_RUNG
   // the same network as SCL:
   "DB368_M_UNIT_03".M_CODES_UNIT_03.Ack_M621 := "DB3710_U2_F3_GRIPPER".CYL.FULL_CLOSED;
END_REGION

REGION Network 72: M621-FIXTURE 3 GRIPPER CLOSE / M110-AXIAL LOCATOR LOCATE FIXTURE 1
   RUNG wire#powerrail
      Contact( "DB338_EXTENDED_M_CODE_UNIT_03".M_code[621] )
      wire#w1
      I_Contact( "DB368_M_UNIT_03".M_CODES_UNIT_03.Ack_M621 )
      I_Contact( "DB2120_MPP_ITC_IPC".RESET_FAULTS )
      I_Contact( "DB368_M_UNIT_03".M_CODES_UNIT_03.M_RESET_PULSE )
      Coil( "DB368_M_UNIT_03".M_CODES_UNIT_03.M621 )
   END_RUNG
   RUNG wire#powerrail
      Contact( "DB368_M_UNIT_03".M_CODES_UNIT_03.M621 )
   END_RUNG wire#w1
   // the same network as SCL:
   "DB368_M_UNIT_03".M_CODES_UNIT_03.M621 := ("DB338_EXTENDED_M_CODE_UNIT_03".M_code[621] OR "DB368_M_UNIT_03".M_CODES_UNIT_03.M621) AND NOT "DB368_M_UNIT_03".M_CODES_UNIT_03.Ack_M621 AND NOT "DB2120_MPP_ITC_IPC".RESET_FAULTS AND NOT "DB368_M_UNIT_03".M_CODES_UNIT_03.M_RESET_PULSE;
END_REGION

REGION Network 73: ACKNOWLEDGE M622-FIXTURE 3 GRIPPER RETURN (READ-IN DISABLE) / ACKNOWLEDGE M111-AXIAL LOCATOR RETURN FIXTURE 1
   RUNG wire#powerrail
      Contact( "DB3710_U2_F3_GRIPPER".CYL.FULL_OPEN )
      Coil( "DB368_M_UNIT_03".M_CODES_UNIT_03.Ack_M622 )
   END_RUNG
   // the same network as SCL:
   "DB368_M_UNIT_03".M_CODES_UNIT_03.Ack_M622 := "DB3710_U2_F3_GRIPPER".CYL.FULL_OPEN;
END_REGION

REGION Network 74: M622-FIXTURE 3 GRIPPER RETURN (READ-IN DISABLE) / M111-AXIAL LOCATOR RETURN FIXTURE 1
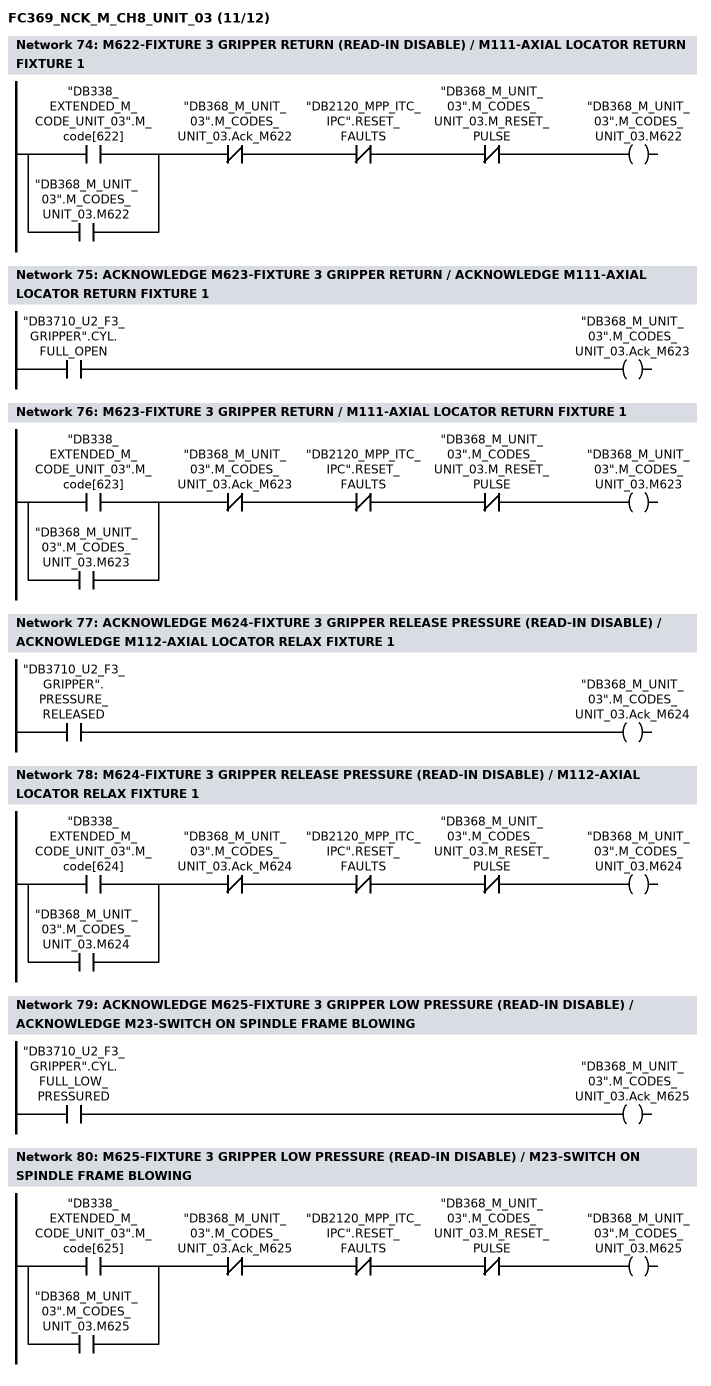
   RUNG wire#powerrail
      Contact( "DB338_EXTENDED_M_CODE_UNIT_03".M_code[622] )
      wire#w1
      I_Contact( "DB368_M_UNIT_03".M_CODES_UNIT_03.Ack_M622 )
      I_Contact( "DB2120_MPP_ITC_IPC".RESET_FAULTS )
      I_Contact( "DB368_M_UNIT_03".M_CODES_UNIT_03.M_RESET_PULSE )
      Coil( "DB368_M_UNIT_03".M_CODES_UNIT_03.M622 )
   END_RUNG
   RUNG wire#powerrail
      Contact( "DB368_M_UNIT_03".M_CODES_UNIT_03.M622 )
   END_RUNG wire#w1
   // the same network as SCL:
   "DB368_M_UNIT_03".M_CODES_UNIT_03.M622 := ("DB338_EXTENDED_M_CODE_UNIT_03".M_code[622] OR "DB368_M_UNIT_03".M_CODES_UNIT_03.M622) AND NOT "DB368_M_UNIT_03".M_CODES_UNIT_03.Ack_M622 AND NOT "DB2120_MPP_ITC_IPC".RESET_FAULTS AND NOT "DB368_M_UNIT_03".M_CODES_UNIT_03.M_RESET_PULSE;
END_REGION

REGION Network 75: ACKNOWLEDGE M623-FIXTURE 3 GRIPPER RETURN / ACKNOWLEDGE M111-AXIAL LOCATOR RETURN FIXTURE 1
   RUNG wire#powerrail
      Contact( "DB3710_U2_F3_GRIPPER".CYL.FULL_OPEN )
      Coil( "DB368_M_UNIT_03".M_CODES_UNIT_03.Ack_M623 )
   END_RUNG
   // the same network as SCL:
   "DB368_M_UNIT_03".M_CODES_UNIT_03.Ack_M623 := "DB3710_U2_F3_GRIPPER".CYL.FULL_OPEN;
END_REGION

REGION Network 76: M623-FIXTURE 3 GRIPPER RETURN / M111-AXIAL LOCATOR RETURN FIXTURE 1
   RUNG wire#powerrail
      Contact( "DB338_EXTENDED_M_CODE_UNIT_03".M_code[623] )
      wire#w1
      I_Contact( "DB368_M_UNIT_03".M_CODES_UNIT_03.Ack_M623 )
      I_Contact( "DB2120_MPP_ITC_IPC".RESET_FAULTS )
      I_Contact( "DB368_M_UNIT_03".M_CODES_UNIT_03.M_RESET_PULSE )
      Coil( "DB368_M_UNIT_03".M_CODES_UNIT_03.M623 )
   END_RUNG
   RUNG wire#powerrail
      Contact( "DB368_M_UNIT_03".M_CODES_UNIT_03.M623 )
   END_RUNG wire#w1
   // the same network as SCL:
   "DB368_M_UNIT_03".M_CODES_UNIT_03.M623 := ("DB338_EXTENDED_M_CODE_UNIT_03".M_code[623] OR "DB368_M_UNIT_03".M_CODES_UNIT_03.M623) AND NOT "DB368_M_UNIT_03".M_CODES_UNIT_03.Ack_M623 AND NOT "DB2120_MPP_ITC_IPC".RESET_FAULTS AND NOT "DB368_M_UNIT_03".M_CODES_UNIT_03.M_RESET_PULSE;
END_REGION

REGION Network 77: ACKNOWLEDGE M624-FIXTURE 3 GRIPPER RELEASE PRESSURE (READ-IN DISABLE) / ACKNOWLEDGE M112-AXIAL LOCATOR RELAX FIXTURE 1
   RUNG wire#powerrail
      Contact( "DB3710_U2_F3_GRIPPER".PRESSURE_RELEASED )
      Coil( "DB368_M_UNIT_03".M_CODES_UNIT_03.Ack_M624 )
   END_RUNG
   // the same network as SCL:
   "DB368_M_UNIT_03".M_CODES_UNIT_03.Ack_M624 := "DB3710_U2_F3_GRIPPER".PRESSURE_RELEASED;
END_REGION

REGION Network 78: M624-FIXTURE 3 GRIPPER RELEASE PRESSURE (READ-IN DISABLE) / M112-AXIAL LOCATOR RELAX FIXTURE 1
   RUNG wire#powerrail
      Contact( "DB338_EXTENDED_M_CODE_UNIT_03".M_code[624] )
      wire#w1
      I_Contact( "DB368_M_UNIT_03".M_CODES_UNIT_03.Ack_M624 )
      I_Contact( "DB2120_MPP_ITC_IPC".RESET_FAULTS )
      I_Contact( "DB368_M_UNIT_03".M_CODES_UNIT_03.M_RESET_PULSE )
      Coil( "DB368_M_UNIT_03".M_CODES_UNIT_03.M624 )
   END_RUNG
   RUNG wire#powerrail
      Contact( "DB368_M_UNIT_03".M_CODES_UNIT_03.M624 )
   END_RUNG wire#w1
   // the same network as SCL:
   "DB368_M_UNIT_03".M_CODES_UNIT_03.M624 := ("DB338_EXTENDED_M_CODE_UNIT_03".M_code[624] OR "DB368_M_UNIT_03".M_CODES_UNIT_03.M624) AND NOT "DB368_M_UNIT_03".M_CODES_UNIT_03.Ack_M624 AND NOT "DB2120_MPP_ITC_IPC".RESET_FAULTS AND NOT "DB368_M_UNIT_03".M_CODES_UNIT_03.M_RESET_PULSE;
END_REGION

REGION Network 79: ACKNOWLEDGE M625-FIXTURE 3 GRIPPER LOW PRESSURE (READ-IN DISABLE) / ACKNOWLEDGE M23-SWITCH ON SPINDLE FRAME BLOWING
   RUNG wire#powerrail
      Contact( "DB3710_U2_F3_GRIPPER".CYL.FULL_LOW_PRESSURED )
      Coil( "DB368_M_UNIT_03".M_CODES_UNIT_03.Ack_M625 )
   END_RUNG
   // the same network as SCL:
   "DB368_M_UNIT_03".M_CODES_UNIT_03.Ack_M625 := "DB3710_U2_F3_GRIPPER".CYL.FULL_LOW_PRESSURED;
END_REGION

REGION Network 80: M625-FIXTURE 3 GRIPPER LOW PRESSURE (READ-IN DISABLE) / M23-SWITCH ON SPINDLE FRAME BLOWING
   RUNG wire#powerrail
      Contact( "DB338_EXTENDED_M_CODE_UNIT_03".M_code[625] )
      wire#w1
      I_Contact( "DB368_M_UNIT_03".M_CODES_UNIT_03.Ack_M625 )
      I_Contact( "DB2120_MPP_ITC_IPC".RESET_FAULTS )
      I_Contact( "DB368_M_UNIT_03".M_CODES_UNIT_03.M_RESET_PULSE )
      Coil( "DB368_M_UNIT_03".M_CODES_UNIT_03.M625 )
   END_RUNG
   RUNG wire#powerrail
      Contact( "DB368_M_UNIT_03".M_CODES_UNIT_03.M625 )
   END_RUNG wire#w1
   // the same network as SCL:
   "DB368_M_UNIT_03".M_CODES_UNIT_03.M625 := ("DB338_EXTENDED_M_CODE_UNIT_03".M_code[625] OR "DB368_M_UNIT_03".M_CODES_UNIT_03.M625) AND NOT "DB368_M_UNIT_03".M_CODES_UNIT_03.Ack_M625 AND NOT "DB2120_MPP_ITC_IPC".RESET_FAULTS AND NOT "DB368_M_UNIT_03".M_CODES_UNIT_03.M_RESET_PULSE;
END_REGION

REGION Network 81: READ-IN DISABLE / Read-in disable
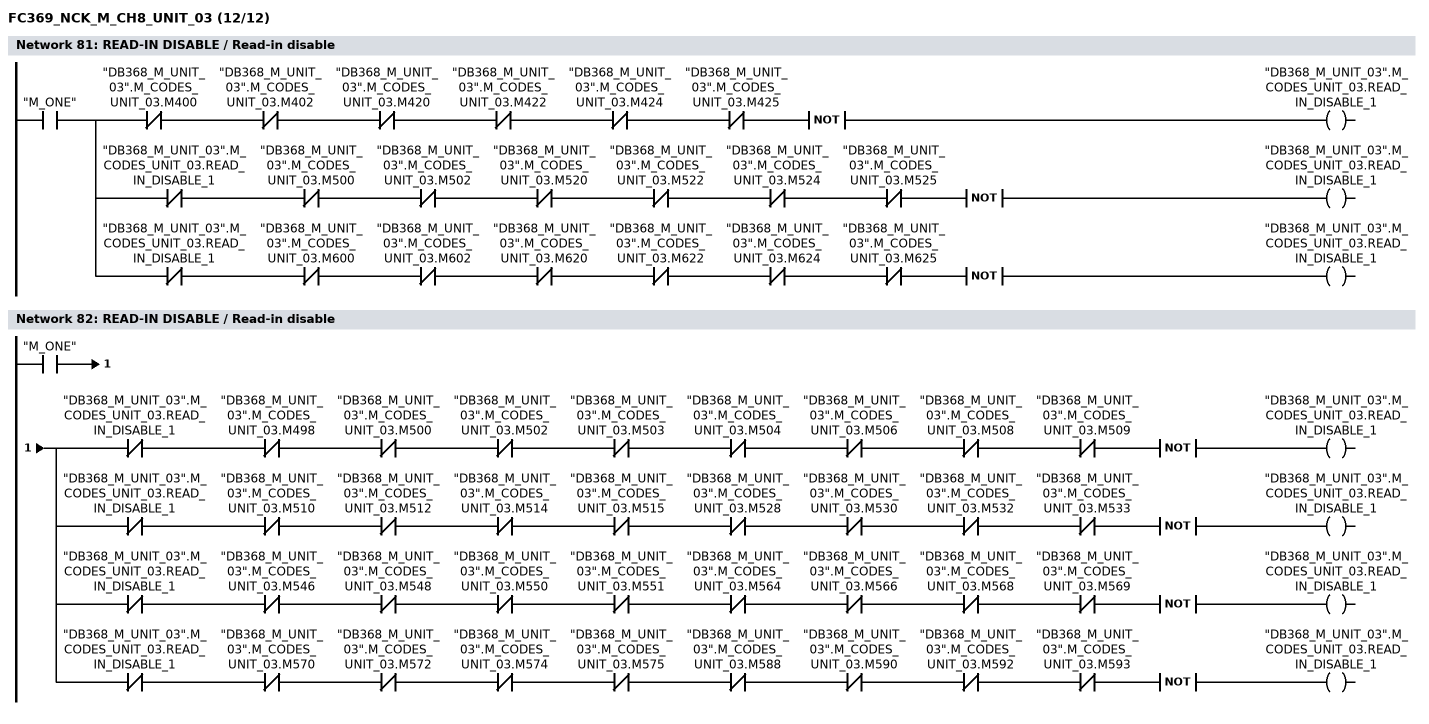
   RUNG wire#powerrail
      Contact( "M_ONE" )
      wire#w1
      I_Contact( "DB368_M_UNIT_03".M_CODES_UNIT_03.M400 )
      I_Contact( "DB368_M_UNIT_03".M_CODES_UNIT_03.M402 )
      I_Contact( "DB368_M_UNIT_03".M_CODES_UNIT_03.M420 )
      I_Contact( "DB368_M_UNIT_03".M_CODES_UNIT_03.M422 )
      I_Contact( "DB368_M_UNIT_03".M_CODES_UNIT_03.M424 )
      I_Contact( "DB368_M_UNIT_03".M_CODES_UNIT_03.M425 )
      Not()
      Coil( "DB368_M_UNIT_03".M_CODES_UNIT_03.READ_IN_DISABLE_1 )
   END_RUNG
   RUNG wire#w1
      I_Contact( "DB368_M_UNIT_03".M_CODES_UNIT_03.READ_IN_DISABLE_1 )
      I_Contact( "DB368_M_UNIT_03".M_CODES_UNIT_03.M500 )
      I_Contact( "DB368_M_UNIT_03".M_CODES_UNIT_03.M502 )
      I_Contact( "DB368_M_UNIT_03".M_CODES_UNIT_03.M520 )
      I_Contact( "DB368_M_UNIT_03".M_CODES_UNIT_03.M522 )
      I_Contact( "DB368_M_UNIT_03".M_CODES_UNIT_03.M524 )
      I_Contact( "DB368_M_UNIT_03".M_CODES_UNIT_03.M525 )
      Not()
      Coil( "DB368_M_UNIT_03".M_CODES_UNIT_03.READ_IN_DISABLE_1 )
   END_RUNG
   RUNG wire#w1
      I_Contact( "DB368_M_UNIT_03".M_CODES_UNIT_03.READ_IN_DISABLE_1 )
      I_Contact( "DB368_M_UNIT_03".M_CODES_UNIT_03.M600 )
      I_Contact( "DB368_M_UNIT_03".M_CODES_UNIT_03.M602 )
      I_Contact( "DB368_M_UNIT_03".M_CODES_UNIT_03.M620 )
      I_Contact( "DB368_M_UNIT_03".M_CODES_UNIT_03.M622 )
      I_Contact( "DB368_M_UNIT_03".M_CODES_UNIT_03.M624 )
      I_Contact( "DB368_M_UNIT_03".M_CODES_UNIT_03.M625 )
      Not()
      Coil( "DB368_M_UNIT_03".M_CODES_UNIT_03.READ_IN_DISABLE_1 )
   END_RUNG
   // the same network as SCL:
   "DB368_M_UNIT_03".M_CODES_UNIT_03.READ_IN_DISABLE_1 := NOT ("M_ONE" AND NOT "DB368_M_UNIT_03".M_CODES_UNIT_03.M400 AND NOT "DB368_M_UNIT_03".M_CODES_UNIT_03.M402 AND NOT "DB368_M_UNIT_03".M_CODES_UNIT_03.M420 AND NOT "DB368_M_UNIT_03".M_CODES_UNIT_03.M422 AND NOT "DB368_M_UNIT_03".M_CODES_UNIT_03.M424 AND NOT "DB368_M_UNIT_03".M_CODES_UNIT_03.M425);
   "DB368_M_UNIT_03".M_CODES_UNIT_03.READ_IN_DISABLE_1 := NOT ("M_ONE" AND NOT "DB368_M_UNIT_03".M_CODES_UNIT_03.READ_IN_DISABLE_1 AND NOT "DB368_M_UNIT_03".M_CODES_UNIT_03.M500 AND NOT "DB368_M_UNIT_03".M_CODES_UNIT_03.M502 AND NOT "DB368_M_UNIT_03".M_CODES_UNIT_03.M520 AND NOT "DB368_M_UNIT_03".M_CODES_UNIT_03.M522 AND NOT "DB368_M_UNIT_03".M_CODES_UNIT_03.M524 AND NOT "DB368_M_UNIT_03".M_CODES_UNIT_03.M525);
   "DB368_M_UNIT_03".M_CODES_UNIT_03.READ_IN_DISABLE_1 := NOT ("M_ONE" AND NOT "DB368_M_UNIT_03".M_CODES_UNIT_03.READ_IN_DISABLE_1 AND NOT "DB368_M_UNIT_03".M_CODES_UNIT_03.M600 AND NOT "DB368_M_UNIT_03".M_CODES_UNIT_03.M602 AND NOT "DB368_M_UNIT_03".M_CODES_UNIT_03.M620 AND NOT "DB368_M_UNIT_03".M_CODES_UNIT_03.M622 AND NOT "DB368_M_UNIT_03".M_CODES_UNIT_03.M624 AND NOT "DB368_M_UNIT_03".M_CODES_UNIT_03.M625);
END_REGION

REGION Network 82: READ-IN DISABLE / Read-in disable
   RUNG wire#powerrail
      Contact( "M_ONE" )
      wire#w1
      I_Contact( "DB368_M_UNIT_03".M_CODES_UNIT_03.READ_IN_DISABLE_1 )
      I_Contact( "DB368_M_UNIT_03".M_CODES_UNIT_03.M498 )
      I_Contact( "DB368_M_UNIT_03".M_CODES_UNIT_03.M500 )
      I_Contact( "DB368_M_UNIT_03".M_CODES_UNIT_03.M502 )
      I_Contact( "DB368_M_UNIT_03".M_CODES_UNIT_03.M503 )
      I_Contact( "DB368_M_UNIT_03".M_CODES_UNIT_03.M504 )
      I_Contact( "DB368_M_UNIT_03".M_CODES_UNIT_03.M506 )
      I_Contact( "DB368_M_UNIT_03".M_CODES_UNIT_03.M508 )
      I_Contact( "DB368_M_UNIT_03".M_CODES_UNIT_03.M509 )
      Not()
      Coil( "DB368_M_UNIT_03".M_CODES_UNIT_03.READ_IN_DISABLE_1 )
   END_RUNG
   RUNG wire#w1
      I_Contact( "DB368_M_UNIT_03".M_CODES_UNIT_03.READ_IN_DISABLE_1 )
      I_Contact( "DB368_M_UNIT_03".M_CODES_UNIT_03.M510 )
      I_Contact( "DB368_M_UNIT_03".M_CODES_UNIT_03.M512 )
      I_Contact( "DB368_M_UNIT_03".M_CODES_UNIT_03.M514 )
      I_Contact( "DB368_M_UNIT_03".M_CODES_UNIT_03.M515 )
      I_Contact( "DB368_M_UNIT_03".M_CODES_UNIT_03.M528 )
      I_Contact( "DB368_M_UNIT_03".M_CODES_UNIT_03.M530 )
      I_Contact( "DB368_M_UNIT_03".M_CODES_UNIT_03.M532 )
      I_Contact( "DB368_M_UNIT_03".M_CODES_UNIT_03.M533 )
      Not()
      Coil( "DB368_M_UNIT_03".M_CODES_UNIT_03.READ_IN_DISABLE_1 )
   END_RUNG
   RUNG wire#w1
      I_Contact( "DB368_M_UNIT_03".M_CODES_UNIT_03.READ_IN_DISABLE_1 )
      I_Contact( "DB368_M_UNIT_03".M_CODES_UNIT_03.M546 )
      I_Contact( "DB368_M_UNIT_03".M_CODES_UNIT_03.M548 )
      I_Contact( "DB368_M_UNIT_03".M_CODES_UNIT_03.M550 )
      I_Contact( "DB368_M_UNIT_03".M_CODES_UNIT_03.M551 )
      I_Contact( "DB368_M_UNIT_03".M_CODES_UNIT_03.M564 )
      I_Contact( "DB368_M_UNIT_03".M_CODES_UNIT_03.M566 )
      I_Contact( "DB368_M_UNIT_03".M_CODES_UNIT_03.M568 )
      I_Contact( "DB368_M_UNIT_03".M_CODES_UNIT_03.M569 )
      Not()
      Coil( "DB368_M_UNIT_03".M_CODES_UNIT_03.READ_IN_DISABLE_1 )
   END_RUNG
   RUNG wire#w1
      I_Contact( "DB368_M_UNIT_03".M_CODES_UNIT_03.READ_IN_DISABLE_1 )
      I_Contact( "DB368_M_UNIT_03".M_CODES_UNIT_03.M570 )
      I_Contact( "DB368_M_UNIT_03".M_CODES_UNIT_03.M572 )
      I_Contact( "DB368_M_UNIT_03".M_CODES_UNIT_03.M574 )
      I_Contact( "DB368_M_UNIT_03".M_CODES_UNIT_03.M575 )
      I_Contact( "DB368_M_UNIT_03".M_CODES_UNIT_03.M588 )
      I_Contact( "DB368_M_UNIT_03".M_CODES_UNIT_03.M590 )
      I_Contact( "DB368_M_UNIT_03".M_CODES_UNIT_03.M592 )
      I_Contact( "DB368_M_UNIT_03".M_CODES_UNIT_03.M593 )
      Not()
      Coil( "DB368_M_UNIT_03".M_CODES_UNIT_03.READ_IN_DISABLE_1 )
   END_RUNG
   // the same network as SCL:
   "DB368_M_UNIT_03".M_CODES_UNIT_03.READ_IN_DISABLE_1 := NOT ("M_ONE" AND NOT "DB368_M_UNIT_03".M_CODES_UNIT_03.READ_IN_DISABLE_1 AND NOT "DB368_M_UNIT_03".M_CODES_UNIT_03.M498 AND NOT "DB368_M_UNIT_03".M_CODES_UNIT_03.M500 AND NOT "DB368_M_UNIT_03".M_CODES_UNIT_03.M502 AND NOT "DB368_M_UNIT_03".M_CODES_UNIT_03.M503 AND NOT "DB368_M_UNIT_03".M_CODES_UNIT_03.M504 AND NOT "DB368_M_UNIT_03".M_CODES_UNIT_03.M506 AND NOT "DB368_M_UNIT_03".M_CODES_UNIT_03.M508 AND NOT "DB368_M_UNIT_03".M_CODES_UNIT_03.M509);
   "DB368_M_UNIT_03".M_CODES_UNIT_03.READ_IN_DISABLE_1 := NOT ("M_ONE" AND NOT "DB368_M_UNIT_03".M_CODES_UNIT_03.READ_IN_DISABLE_1 AND NOT "DB368_M_UNIT_03".M_CODES_UNIT_03.M510 AND NOT "DB368_M_UNIT_03".M_CODES_UNIT_03.M512 AND NOT "DB368_M_UNIT_03".M_CODES_UNIT_03.M514 AND NOT "DB368_M_UNIT_03".M_CODES_UNIT_03.M515 AND NOT "DB368_M_UNIT_03".M_CODES_UNIT_03.M528 AND NOT "DB368_M_UNIT_03".M_CODES_UNIT_03.M530 AND NOT "DB368_M_UNIT_03".M_CODES_UNIT_03.M532 AND NOT "DB368_M_UNIT_03".M_CODES_UNIT_03.M533);
   "DB368_M_UNIT_03".M_CODES_UNIT_03.READ_IN_DISABLE_1 := NOT ("M_ONE" AND NOT "DB368_M_UNIT_03".M_CODES_UNIT_03.READ_IN_DISABLE_1 AND NOT "DB368_M_UNIT_03".M_CODES_UNIT_03.M546 AND NOT "DB368_M_UNIT_03".M_CODES_UNIT_03.M548 AND NOT "DB368_M_UNIT_03".M_CODES_UNIT_03.M550 AND NOT "DB368_M_UNIT_03".M_CODES_UNIT_03.M551 AND NOT "DB368_M_UNIT_03".M_CODES_UNIT_03.M564 AND NOT "DB368_M_UNIT_03".M_CODES_UNIT_03.M566 AND NOT "DB368_M_UNIT_03".M_CODES_UNIT_03.M568 AND NOT "DB368_M_UNIT_03".M_CODES_UNIT_03.M569);
   "DB368_M_UNIT_03".M_CODES_UNIT_03.READ_IN_DISABLE_1 := NOT ("M_ONE" AND NOT "DB368_M_UNIT_03".M_CODES_UNIT_03.READ_IN_DISABLE_1 AND NOT "DB368_M_UNIT_03".M_CODES_UNIT_03.M570 AND NOT "DB368_M_UNIT_03".M_CODES_UNIT_03.M572 AND NOT "DB368_M_UNIT_03".M_CODES_UNIT_03.M574 AND NOT "DB368_M_UNIT_03".M_CODES_UNIT_03.M575 AND NOT "DB368_M_UNIT_03".M_CODES_UNIT_03.M588 AND NOT "DB368_M_UNIT_03".M_CODES_UNIT_03.M590 AND NOT "DB368_M_UNIT_03".M_CODES_UNIT_03.M592 AND NOT "DB368_M_UNIT_03".M_CODES_UNIT_03.M593);
END_REGION
END_FUNCTION
